KUKA KRL program: MyProgram_323().src

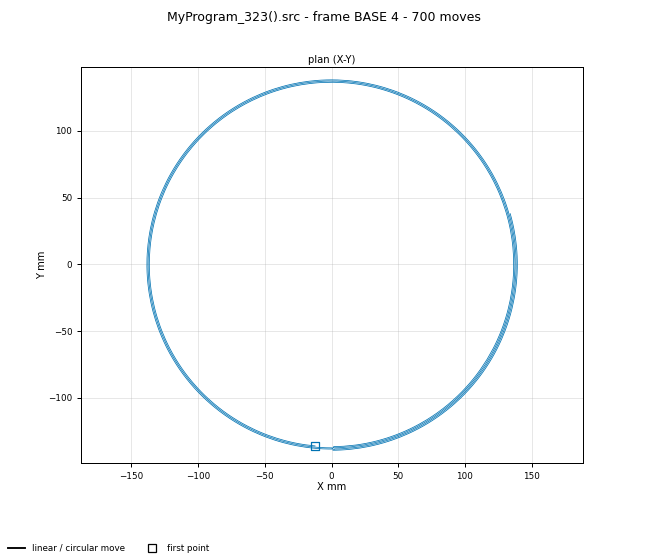
[picture p0: tool path of MyProgram_323().src in frame BASE 4, 700 of 700 moves have a stored position in this frame; points joined in program order, loops and branches not executed]
&ACCESS RVP
&REL 1
&PARAM TEMPLATE = C:\KRC\Roboter\Template\vorgabe
&PARAM EDITMASK = *
DEF MyProgram_323()
; ---- Setting reference (Base) ----
$BASE = BASE_DATA[4]

; --------------------------
; ---- Setting tool (TCP) ----
$TOOL = TOOL_DATA[3]
; --------------------------

$VEL.CP = VEL_APROX_PRINT
Startdeposition()
$VEL.CP = VEL_PRINT
LIN {X -12.3111,Y -135.9679,Z 186,A -89.4743,B 2.9889,C 0.3145,E1 2.9942,E2 182.4213} C_DIS
LIN {X -19.238,Y -135.1598,Z 186,A -92.5323,B 2.9889,C 0.3149,E1 2.9856,E2 185.4978} C_DIS
LIN {X -23.7694,Y -134.4372,Z 186,A -94.3944,B 2.9889,C 0.3139,E1 2.9805,E2 187.3522} C_DIS
LIN {X -27.1514,Y -133.7948,Z 186,A -95.8563,B 2.9889,C 0.3134,E1 2.9765,E2 188.8169} C_DIS
LIN {X -30.8353,Y -132.9948,Z 186,A -97.5736,B 2.9889,C 0.3136,E1 2.9718,E2 190.5525} C_DIS
LIN {X -35.0308,Y -131.9511,Z 186,A -99.2612,B 2.9891,C 0.3118,E1 2.9672,E2 192.2239} C_DIS
LIN {X -38.3777,Y -131.0167,Z 186,A -100.6732,B 2.9893,C 0.3107,E1 2.9634,E2 193.6301} C_DIS
LIN {X -41.0826,Y -130.1947,Z 186,A -101.9812,B 2.9893,C 0.3107,E1 2.9599,E2 194.9545} C_DIS
LIN {X -44.5379,Y -129.0528,Z 186,A -103.3999,B 2.9895,C 0.3088,E1 2.9562,E2 196.3593} C_DIS
LIN {X -47.6308,Y -127.9436,Z 186,A -104.8022,B 2.9895,C 0.3079,E1 2.9525,E2 197.7649} C_DIS
LIN {X -50.8322,Y -126.7057,Z 186,A -106.3845,B 2.9895,C 0.3074,E1 2.9483,E2 199.3662} C_DIS
LIN {X -54.0849,Y -125.3516,Z 186,A -107.898,B 2.9897,C 0.3062,E1 2.9444,E2 200.8845} C_DIS
LIN {X -57.3156,Y -123.9076,Z 186,A -109.3363,B 2.9899,C 0.3045,E1 2.9408,E2 202.3169} C_DIS
LIN {X -60.3748,Y -122.4461,Z 186,A -110.745,B 2.9901,C 0.3028,E1 2.9372,E2 203.724} C_DIS
LIN {X -63.188,Y -121.0188,Z 186,A -112.1763,B 2.9901,C 0.3019,E1 2.9336,E2 205.1695} C_DIS
LIN {X -67.1147,Y -118.8882,Z 186,A -113.9223,B 2.9905,C 0.2989,E1 2.9294,E2 206.8989} C_DIS
LIN {X -70.3666,Y -116.993,Z 186,A -115.791,B 2.9905,C 0.2985,E1 2.9248,E2 208.8057} C_DIS
LIN {X -74.0884,Y -114.6722,Z 186,A -117.6408,B 2.9908,C 0.296,E1 2.9204,E2 210.6567} C_DIS
LIN {X -77.5445,Y -112.3641,Z 186,A -119.4603,B 2.991,C 0.2938,E1 2.9162,E2 212.4861} C_DIS
LIN {X -81.1661,Y -109.7768,Z 186,A -121.4187,B 2.9912,C 0.2914,E1 2.9117,E2 214.4563} C_DIS
LIN {X -84.7687,Y -107.0191,Z 186,A -123.3765,B 2.9915,C 0.2886,E1 2.9074,E2 216.421} C_DIS
LIN {X -88.3206,Y -104.1067,Z 186,A -125.3337,B 2.9918,C 0.2855,E1 2.9032,E2 218.382} C_DIS
LIN {X -91.8517,Y -101.005,Z 186,A -127.3307,B 2.9921,C 0.2821,E1 2.899,E2 220.382} C_DIS
LIN {X -95.064,Y -97.9876,Z 186,A -129.1105,B 2.9924,C 0.2784,E1 2.8955,E2 222.1525} C_DIS
LIN {X -97.6899,Y -95.3703,Z 186,A -130.752,B 2.9927,C 0.2758,E1 2.8922,E2 223.8048} C_DIS
LIN {X -100.5401,Y -92.3602,Z 186,A -132.7985,B 2.9929,C 0.2738,E1 2.8882,E2 225.8909} C_DIS
LIN {X -103.9141,Y -88.5472,Z 186,A -134.8828,B 2.9933,C 0.2692,E1 2.8844,E2 227.9679} C_DIS
LIN {X -106.7399,Y -85.1195,Z 186,A -136.8215,B 2.9936,C 0.2656,E1 2.881,E2 229.9159} C_DIS
LIN {X -109.4795,Y -81.5656,Z 186,A -138.7616,B 2.9939,C 0.2618,E1 2.8777,E2 231.8628} C_DIS
LIN {X -112.1537,Y -77.8479,Z 186,A -140.7582,B 2.9943,C 0.2578,E1 2.8745,E2 233.8686} C_DIS
LIN {X -114.7019,Y -74.0428,Z 186,A -142.7414,B 2.9946,C 0.2537,E1 2.8714,E2 235.8592} C_DIS
LIN {X -117.0022,Y -70.3515,Z 186,A -144.5127,B 2.995,C 0.2492,E1 2.8688,E2 237.623} C_DIS
LIN {X -119.2801,Y -66.4159,Z 186,A -146.6652,B 2.9953,C 0.2456,E1 2.8658,E2 239.8061} C_DIS
LIN {X -121.5017,Y -62.2546,Z 186,A -148.7079,B 2.9957,C 0.241,E1 2.8631,E2 241.8562} C_DIS
LIN {X -123.127,Y -58.9739,Z 186,A -150.2353,B 2.996,C 0.2371,E1 2.8613,E2 243.3817} C_DIS
LIN {X -124.5737,Y -55.8532,Z 186,A -151.7312,B 2.9963,C 0.2337,E1 2.8595,E2 244.8838} C_DIS
LIN {X -125.921,Y -52.7458,Z 186,A -153.201,B 2.9965,C 0.2303,E1 2.8579,E2 246.3591} C_DIS
LIN {X -127.1093,Y -49.8151,Z 186,A -154.433,B 2.9968,C 0.2265,E1 2.8566,E2 247.5785} C_DIS
LIN {X -128.3866,Y -46.423,Z 186,A -156.1533,B 2.9971,C 0.2233,E1 2.8549,E2 249.3235} C_DIS
LIN {X -130.7067,Y -39.4242,Z 186,A -159.5632,B 2.9976,C 0.2162,E1 2.852,E2 252.7722} C_DIS
LIN {X -131.5486,Y -36.5137,Z 186,A -160.8706,B 2.9978,C 0.2129,E1 2.851,E2 254.0835} C_DIS
LIN {X -132.6266,Y -32.3816,Z 186,A -162.7159,B 2.9981,C 0.2082,E1 2.8497,E2 255.9346} C_DIS
LIN {X -133.4322,Y -28.8806,Z 186,A -164.1633,B 2.9984,C 0.2039,E1 2.8488,E2 257.3735} C_DIS
LIN {X -134.0497,Y -25.8648,Z 186,A -165.6158,B 2.9986,C 0.2009,E1 2.848,E2 258.8457} C_DIS
LIN {X -134.6734,Y -22.3906,Z 186,A -167.1966,B 2.9989,C 0.1972,E1 2.8473,E2 260.4382} C_DIS
LIN {X -135.3221,Y -18.0645,Z 186,A -169.1058,B 2.9992,C 0.1923,E1 2.8465,E2 262.3556} C_DIS
LIN {X -135.7244,Y -14.737,Z 186,A -170.6184,B 2.9994,C 0.1888,E1 2.846,E2 263.8807} C_DIS
LIN {X -136.1225,Y -10.4513,Z 186,A -172.5183,B 2.9997,C 0.184,E1 2.8456,E2 265.7912} C_DIS
LIN {X -136.3524,Y -6.8079,Z 186,A -174.1089,B 3,C 0.1799,E1 2.8453,E2 267.3882} C_DIS
LIN {X -136.4965,Y -2.6863,Z 186,A -175.9244,B 3.0002,C 0.1754,E1 2.8452,E2 269.2133} C_DIS
LIN {X -136.5203,Y 0.8769,Z 186,A -177.5554,B 3.0005,C 0.1716,E1 2.8452,E2 270.8603} C_DIS
LIN {X -136.4303,Y 5.0183,Z 186,A -179.3071,B 3.0007,C 0.1668,E1 2.8453,E2 272.6124} C_DIS
LIN {X -136.2757,Y 8.2022,Z 186,A 179.3242,B 3.0009,C 0.1631,E1 2.8455,E2 273.9841} C_DIS
LIN {X -136.0283,Y 11.6019,Z 186,A 177.7468,B 3.0011,C 0.1596,E1 2.8459,E2 275.5788} C_DIS
LIN {X -135.6057,Y 15.7966,Z 186,A 175.8905,B 3.0014,C 0.1549,E1 2.8464,E2 277.4448} C_DIS
LIN {X -135.1037,Y 19.6307,Z 186,A 174.1589,B 3.0016,C 0.1508,E1 2.8471,E2 279.1888} C_DIS
LIN {X -134.4438,Y 23.7324,Z 186,A 172.4562,B 3.0018,C 0.1458,E1 2.8479,E2 280.8851} C_DIS
LIN {X -133.8588,Y 26.8368,Z 186,A 170.5174,B 3.0018,C 0.1442,E1 2.849,E2 282.8987} C_DIS
LIN {X -132.936,Y 31.0929,Z 186,A 168.9702,B 3.0022,C 0.1382,E1 2.8499,E2 284.4101} C_DIS
LIN {X -131.9802,Y 34.9217,Z 186,A 167.2952,B 3.0024,C 0.1338,E1 2.8511,E2 286.0861} C_DIS
LIN {X -131.1717,Y 37.8484,Z 186,A 165.5608,B 3.0024,C 0.1319,E1 2.8525,E2 287.8762} C_DIS
LIN {X -129.9932,Y 41.7134,Z 186,A 164.2257,B 3.0027,C 0.1261,E1 2.8536,E2 289.1657} C_DIS
LIN {X -129.1127,Y 44.3649,Z 186,A 162.8354,B 3.0028,C 0.1238,E1 2.8548,E2 290.5819} C_DIS
LIN {X -127.3868,Y 49.1014,Z 186,A 160.7805,B 3.003,C 0.118,E1 2.8568,E2 292.6278} C_DIS
LIN {X -124.8679,Y 55.1955,Z 186,A 157.597,B 3.0033,C 0.1124,E1 2.8604,E2 295.8601} C_DIS
LIN {X -123.4731,Y 58.2496,Z 186,A 156.3105,B 3.0033,C 0.1083,E1 2.8619,E2 297.1306} C_DIS
LIN {X -121.8264,Y 61.6167,Z 186,A 154.8044,B 3.0035,C 0.1042,E1 2.8637,E2 298.6272} C_DIS
LIN {X -120.0726,Y 64.9727,Z 186,A 153.0054,B 3.0037,C 0.101,E1 2.8661,E2 300.4508} C_DIS
LIN {X -117.8522,Y 68.9177,Z 186,A 151.0476,B 3.0037,C 0.0966,E1 2.8689,E2 302.4141} C_DIS
LIN {X -115.5398,Y 72.7277,Z 186,A 149.3838,B 3.004,C 0.0914,E1 2.8713,E2 304.0513} C_DIS
LIN {X -112.8554,Y 76.8272,Z 186,A 146.5212,B 3.004,C 0.0898,E1 2.8759,E2 307.0099} C_DIS
LIN {X -110.2473,Y 80.5257,Z 186,A 144.9632,B 3.0042,C 0.0842,E1 2.8783,E2 308.5255} C_DIS
LIN {X -108.0587,Y 83.4392,Z 186,A 142.6585,B 3.0042,C 0.0839,E1 2.8825,E2 310.9221} C_DIS
LIN {X -104.259,Y 88.1412,Z 186,A 140.5187,B 3.0044,C 0.0769,E1 2.8862,E2 313.0125} C_DIS
LIN {X -101.9478,Y 90.8048,Z 186,A 139.2264,B 3.0044,C 0.0731,E1 2.8885,E2 314.2811} C_DIS
LIN {X -98.977,Y 94.0341,Z 186,A 137.3781,B 3.0045,C 0.0695,E1 2.8921,E2 316.1288} C_DIS
LIN {X -95.5224,Y 97.5407,Z 186,A 135.1953,B 3.0046,C 0.066,E1 2.8964,E2 318.3242} C_DIS
LIN {X -92.1681,Y 100.7167,Z 186,A 133.1879,B 3.0046,C 0.0627,E1 2.9005,E2 320.3384} C_DIS
LIN {X -88.7865,Y 103.7103,Z 186,A 131.2058,B 3.0048,C 0.0597,E1 2.9047,E2 322.3296} C_DIS
LIN {X -86.4597,Y 105.6572,Z 186,A 129.1909,B 3.0048,C 0.0608,E1 2.9093,E2 324.4318} C_DIS
LIN {X -81.7175,Y 109.3665,Z 186,A 127.307,B 3.0048,C 0.0538,E1 2.9133,E2 326.2376} C_DIS
LIN {X -78.0842,Y 111.9893,Z 186,A 125.4022,B 3.0049,C 0.051,E1 2.9176,E2 328.1439} C_DIS
LIN {X -74.4651,Y 114.4277,Z 186,A 123.4234,B 3.0049,C 0.049,E1 2.9223,E2 330.139} C_DIS
LIN {X -69.1963,Y 117.6886,Z 186,A 120.8537,B 3.005,C 0.0453,E1 2.9284,E2 332.7033} C_DIS
LIN {X -64.6844,Y 120.2276,Z 186,A 117.9757,B 3.005,C 0.046,E1 2.9357,E2 335.6634} C_DIS
LIN {X -59.6478,Y 122.8047,Z 186,A 116.2676,B 3.005,C 0.04,E1 2.9398,E2 337.2911} C_DIS
LIN {X -56.2549,Y 124.394,Z 186,A 114.6333,B 3.0051,C 0.0386,E1 2.9439,E2 338.9317} C_DIS
LIN {X -53.3798,Y 125.6562,Z 186,A 112.5963,B 3.0051,C 0.041,E1 2.9494,E2 341.0531} C_DIS
LIN {X -48.161,Y 127.745,Z 186,A 110.9689,B 3.0051,C 0.035,E1 2.9534,E2 342.5924} C_DIS
LIN {X -44.7133,Y 128.9919,Z 186,A 109.423,B 3.0051,C 0.0338,E1 2.9575,E2 344.1382} C_DIS
LIN {X -41.5386,Y 130.0491,Z 186,A 108.0354,B 3.0051,C 0.0326,E1 2.9612,E2 345.523} C_DIS
LIN {X -37.3561,Y 131.313,Z 186,A 105.9999,B 3.0051,C 0.0325,E1 2.9667,E2 347.5815} C_DIS
LIN {X -33.3708,Y 132.3808,Z 186,A 104.3549,B 3.0051,C 0.031,E1 2.9711,E2 349.2152} C_DIS
LIN {X -29.3101,Y 133.3395,Z 186,A 102.5381,B 3.0051,C 0.0305,E1 2.9761,E2 351.0389} C_DIS
LIN {X -25.8157,Y 134.0591,Z 186,A 101.1794,B 3.0052,C 0.029,E1 2.9798,E2 352.3802} C_DIS
LIN {X -22.6569,Y 134.629,Z 186,A 99.7557,B 3.0052,C 0.029,E1 2.9837,E2 353.8124} C_DIS
LIN {X -19.1156,Y 135.1773,Z 186,A 98.1668,B 3.0052,C 0.029,E1 2.9881,E2 355.4106} C_DIS
LIN {X -15.9064,Y 135.5925,Z 186,A 96.2554,B 3.0052,C 0.0321,E1 2.9936,E2 357.3868} C_DIS
LIN {X -10.8726,Y 136.0899,Z 186,A 94.9122,B 3.0052,C 0.0271,E1 2.9971,E2 358.6368} C_DIS
LIN {X -6.7864,Y 136.3535,Z 186,A 92.9753,B 3.0052,C 0.0284,E1 3.0026,E2 360.5989} C_DIS
LIN {X 1.2265,Y 136.5176,Z 186,A 89.7328,B 3.0052,C 0.0279,E1 3.0116,E2 363.8257} C_DIS
LIN {X 7.1604,Y 136.3347,Z 186,A 87.0766,B 3.0052,C 0.0296,E1 3.0191,E2 366.5005} C_DIS
LIN {X 12.8357,Y 135.9176,Z 186,A 84.5619,B 3.0052,C 0.0312,E1 3.0261,E2 369.0293} C_DIS
LIN {X 18.3432,Y 135.2855,Z 186,A 82.3763,B 3.0052,C 0.0314,E1 3.0321,E2 371.1974} C_DIS
LIN {X 22.0077,Y 134.7373,Z 186,A 80.9108,B 3.0052,C 0.0316,E1 3.0361,E2 372.6518} C_DIS
LIN {X 25.5439,Y 134.111,Z 186,A 79.4605,B 3.0052,C 0.0322,E1 3.0401,E2 374.0947} C_DIS
LIN {X 29.2124,Y 133.3606,Z 186,A 77.8146,B 3.0052,C 0.0338,E1 3.0446,E2 375.749} C_DIS
LIN {X 33.2752,Y 132.405,Z 186,A 76.1571,B 3.0052,C 0.0345,E1 3.0491,E2 377.3949} C_DIS
LIN {X 36.6894,Y 131.4995,Z 186,A 74.7084,B 3.0052,C 0.0355,E1 3.053,E2 378.8391} C_DIS
LIN {X 40.0511,Y 130.5149,Z 186,A 73.3177,B 3.0052,C 0.0363,E1 3.0567,E2 380.22} C_DIS
LIN {X 43.289,Y 129.477,Z 186,A 71.8669,B 3.0052,C 0.0379,E1 3.0606,E2 381.6734} C_DIS
LIN {X 46.795,Y 128.2525,Z 186,A 70.2657,B 3.0051,C 0.0399,E1 3.0648,E2 383.2794} C_DIS
LIN {X 50.596,Y 126.8009,Z 186,A 68.7271,B 3.0051,C 0.0405,E1 3.0687,E2 384.7975} C_DIS
LIN {X 53.9337,Y 125.4169,Z 186,A 67.2445,B 3.0051,C 0.0421,E1 3.0726,E2 386.2757} C_DIS
LIN {X 57.0285,Y 124.0404,Z 186,A 65.7416,B 3.0051,C 0.0445,E1 3.0764,E2 387.7883} C_DIS
LIN {X 60.1298,Y 122.5669,Z 186,A 64.3487,B 3.005,C 0.046,E1 3.0799,E2 389.1752} C_DIS
LIN {X 63.3023,Y 120.9587,Z 186,A 62.9182,B 3.005,C 0.0476,E1 3.0834,E2 390.5981} C_DIS
LIN {X 67.5166,Y 118.6603,Z 186,A 60.8638,B 3.005,C 0.0509,E1 3.0885,E2 392.6573} C_DIS
LIN {X 71.4257,Y 116.349,Z 186,A 59.0755,B 3.0049,C 0.0529,E1 3.0927,E2 394.4313} C_DIS
LIN {X 74.975,Y 114.0942,Z 186,A 57.2858,B 3.0049,C 0.0559,E1 3.0969,E2 396.224} C_DIS
LIN {X 78.8427,Y 111.4566,Z 186,A 55.4054,B 3.0048,C 0.0585,E1 3.1012,E2 398.0942} C_DIS
LIN {X 82.5066,Y 108.7726,Z 186,A 53.5229,B 3.0048,C 0.0617,E1 3.1054,E2 399.9739} C_DIS
LIN {X 86.0456,Y 105.9956,Z 186,A 51.6692,B 3.0047,C 0.0649,E1 3.1095,E2 401.8236} C_DIS
LIN {X 89.4469,Y 103.1414,Z 186,A 49.8729,B 3.0046,C 0.0678,E1 3.1133,E2 403.6119} C_DIS
LIN {X 95.1093,Y 97.9437,Z 186,A 46.7896,B 3.0045,C 0.073,E1 3.1196,E2 406.6783} C_DIS
LIN {X 97.8786,Y 95.1766,Z 186,A 44.8441,B 3.0043,C 0.079,E1 3.1234,E2 408.6608} C_DIS
LIN {X 100.6933,Y 92.1935,Z 186,A 43.5559,B 3.0043,C 0.0789,E1 3.1258,E2 409.8967} C_DIS
LIN {X 103.6368,Y 88.8719,Z 186,A 41.7233,B 3.0043,C 0.0827,E1 3.1291,E2 411.7259} C_DIS
LIN {X 106.4156,Y 85.5248,Z 186,A 39.9701,B 3.0041,C 0.0861,E1 3.1322,E2 413.4707} C_DIS
LIN {X 109.1359,Y 82.0252,Z 186,A 38.179,B 3.0041,C 0.0897,E1 3.1352,E2 415.2538} C_DIS
LIN {X 111.7542,Y 78.4208,Z 186,A 36.3595,B 3.0039,C 0.0936,E1 3.1382,E2 417.0677} C_DIS
LIN {X 113.7016,Y 75.5694,Z 186,A 34.9815,B 3.0039,C 0.0964,E1 3.1403,E2 418.4373} C_DIS
LIN {X 116.1565,Y 71.7395,Z 186,A 32.9663,B 3.0036,C 0.102,E1 3.1433,E2 420.4662} C_DIS
LIN {X 119.222,Y 66.5209,Z 186,A 30.6725,B 3.0035,C 0.106,E1 3.1465,E2 422.7306} C_DIS
LIN {X 121.467,Y 62.3227,Z 186,A 28.9267,B 3.0034,C 0.1087,E1 3.1487,E2 424.4458} C_DIS
LIN {X 123.0445,Y 59.1467,Z 186,A 27.6386,B 3.0034,C 0.1106,E1 3.1503,E2 425.7097} C_DIS
LIN {X 124.2101,Y 56.6613,Z 186,A 26.2314,B 3.0031,C 0.116,E1 3.152,E2 427.1491} C_DIS
LIN {X 125.8549,Y 52.904,Z 186,A 24.7918,B 3.0031,C 0.1178,E1 3.1535,E2 428.5544} C_DIS
LIN {X 128.2307,Y 46.8553,Z 186,A 22.0445,B 3.0027,C 0.1252,E1 3.1563,E2 431.3054} C_DIS
LIN {X 129.4084,Y 43.4949,Z 186,A 20.6357,B 3.0027,C 0.1284,E1 3.1575,E2 432.7043} C_DIS
LIN {X 130.4095,Y 40.3955,Z 186,A 19.2687,B 3.0024,C 0.1321,E1 3.1587,E2 434.0719} C_DIS
LIN {X 131.4793,Y 36.7617,Z 186,A 17.7861,B 3.0024,C 0.1354,E1 3.1598,E2 435.542} C_DIS
LIN {X 132.5414,Y 32.7352,Z 186,A 16.0718,B 3.0021,C 0.1398,E1 3.161,E2 437.2531} C_DIS
LIN {X 133.3882,Y 29.0848,Z 186,A 14.6294,B 3.002,C 0.1429,E1 3.1619,E2 438.68} C_DIS
LIN {X 134.1341,Y 25.4233,Z 186,A 13.1458,B 3.0018,C 0.1464,E1 3.1627,E2 440.1538} C_DIS
LIN {X 134.8123,Y 21.5488,Z 186,A 11.5791,B 3.0016,C 0.1502,E1 3.1634,E2 441.7109} C_DIS
LIN {X 135.2752,Y 18.422,Z 186,A 9.6378,B 3.0011,C 0.1599,E1 3.1642,E2 443.7298} C_DIS
LIN {X 135.9042,Y 12.9748,Z 186,A 8.4515,B 3.0013,C 0.1555,E1 3.1645,E2 444.7776} C_DIS
LIN {X 136.407,Y 5.6162,Z 186,A 5.3662,B 3.0009,C 0.1642,E1 3.1651,E2 447.8638} C_DIS
LIN {X 136.5062,Y -2.0993,Z 186,A 1.3136,B 2.9999,C 0.1812,E1 3.1651,E2 452.0211} C_DIS
LIN {X 136.2808,Y -8.1196,Z 186,A -0.3193,B 2.9999,C 0.1796,E1 3.1648,E2 453.5429} C_DIS
LIN {X 135.9648,Y -12.3354,Z 186,A -2.5049,B 2.9994,C 0.1886,E1 3.1643,E2 455.7818} C_DIS
LIN {X 135.4992,Y -16.6892,Z 186,A -3.8904,B 2.9994,C 0.1894,E1 3.1639,E2 457.1113} C_DIS
LIN {X 134.9309,Y -20.7833,Z 186,A -5.4477,B 2.9992,C 0.1925,E1 3.1632,E2 458.6473} C_DIS
LIN {X 134.3821,Y -24.0773,Z 186,A -6.7467,B 2.999,C 0.1954,E1 3.1626,E2 459.9342} C_DIS
LIN {X 133.7801,Y -27.2236,Z 186,A -7.9962,B 2.9988,C 0.1982,E1 3.162,E2 461.1726} C_DIS
LIN {X 133.149,Y -30.1605,Z 186,A -9.288,B 2.9986,C 0.202,E1 3.1612,E2 462.4692} C_DIS
LIN {X 132.4036,Y -33.2808,Z 186,A -10.5452,B 2.9984,C 0.2048,E1 3.1604,E2 463.716} C_DIS
LIN {X 131.556,Y -36.4873,Z 186,A -11.9479,B 2.9981,C 0.2087,E1 3.1593,E2 465.1211} C_DIS
LIN {X 130.4126,Y -40.3853,Z 186,A -13.5042,B 2.9979,C 0.2119,E1 3.1581,E2 466.6597} C_DIS
LIN {X 128.6481,Y -45.6978,Z 186,A -15.827,B 2.9974,C 0.218,E1 3.156,E2 468.981} C_DIS
LIN {X 127.2845,Y -49.3646,Z 186,A -17.2732,B 2.9973,C 0.2204,E1 3.1546,E2 470.4032} C_DIS
LIN {X 125.978,Y -52.6091,Z 186,A -18.8924,B 2.9969,C 0.2258,E1 3.1529,E2 472.043} C_DIS
LIN {X 124.0407,Y -57.0278,Z 186,A -20.7104,B 2.9966,C 0.229,E1 3.1508,E2 473.8359} C_DIS
LIN {X 122.5799,Y -60.1036,Z 186,A -22.0566,B 2.9964,C 0.2319,E1 3.1492,E2 475.1725} C_DIS
LIN {X 120.9462,Y -63.3261,Z 186,A -23.2628,B 2.9964,C 0.2328,E1 3.1477,E2 476.3398} C_DIS
LIN {X 116.5433,Y -71.109,Z 186,A -27.0396,B 2.9956,C 0.2424,E1 3.1425,E2 480.123} C_DIS
LIN {X 111.4881,Y -78.7982,Z 186,A -30.8987,B 2.9948,C 0.2517,E1 3.1365,E2 483.985} C_DIS
LIN {X 108.7858,Y -82.4892,Z 186,A -32.7657,B 2.9945,C 0.2556,E1 3.1334,E2 485.8467} C_DIS
LIN {X 106.2159,Y -85.7725,Z 186,A -34.4538,B 2.9942,C 0.259,E1 3.1305,E2 487.5282} C_DIS
LIN {X 103.4473,Y -89.0919,Z 186,A -36.1448,B 2.9939,C 0.2619,E1 3.1274,E2 489.2046} C_DIS
LIN {X 100.2325,Y -92.6949,Z 186,A -38.1537,B 2.9936,C 0.2662,E1 3.1237,E2 491.2128} C_DIS
LIN {X 97.6082,Y -95.4536,Z 186,A -40.0748,B 2.993,C 0.2725,E1 3.1199,E2 493.1773} C_DIS
LIN {X 94.4964,Y -98.5353,Z 186,A -41.3875,B 2.993,C 0.2715,E1 3.1174,E2 494.423} C_DIS
LIN {X 90.4497,Y -102.2623,Z 186,A -43.6905,B 2.9927,C 0.276,E1 3.1126,E2 496.7271} C_DIS
LIN {X 87.1048,Y -105.126,Z 186,A -45.9044,B 2.992,C 0.2828,E1 3.1077,E2 498.9902} C_DIS
LIN {X 83.5684,Y -107.9586,Z 186,A -46.982,B 2.9924,C 0.279,E1 3.1056,E2 499.9614} C_DIS
LIN {X 79.133,Y -111.2511,Z 186,A -49.5837,B 2.9918,C 0.2856,E1 3.0997,E2 502.6023} C_DIS
LIN {X 75.5393,Y -113.7217,Z 186,A -51.357,B 2.9915,C 0.2882,E1 3.0956,E2 504.3694} C_DIS
LIN {X 71.532,Y -116.2838,Z 186,A -53.3903,B 2.9912,C 0.2918,E1 3.0907,E2 506.4091} C_DIS
LIN {X 65.5581,Y -119.7535,Z 186,A -56.1325,B 2.9909,C 0.2949,E1 3.0841,E2 509.1329} C_DIS
LIN {X 62.147,Y -121.5565,Z 186,A -57.6033,B 2.9908,C 0.2959,E1 3.0805,E2 510.5852} C_DIS
LIN {X 59.1591,Y -123.0385,Z 186,A -59.0602,B 2.9905,C 0.2983,E1 3.0768,E2 512.0506} C_DIS
LIN {X 55.5909,Y -124.6911,Z 186,A -60.5881,B 2.9905,C 0.2995,E1 3.073,E2 513.5636} C_DIS
LIN {X 52.4141,Y -126.0595,Z 186,A -62.034,B 2.9902,C 0.3012,E1 3.0693,E2 515.0097} C_DIS
LIN {X 48.6609,Y -127.5578,Z 186,A -63.681,B 2.9901,C 0.3028,E1 3.065,E2 516.6515} C_DIS
LIN {X 44.8703,Y -128.9375,Z 186,A -65.3992,B 2.9899,C 0.3049,E1 3.0605,E2 518.374} C_DIS
LIN {X 41.2755,Y -130.1331,Z 186,A -66.9553,B 2.9897,C 0.3062,E1 3.0563,E2 519.9268} C_DIS
LIN {X 37.195,Y -131.3581,Z 186,A -68.7222,B 2.9896,C 0.3077,E1 3.0516,E2 521.6921} C_DIS
LIN {X 33.8183,Y -132.2672,Z 186,A -70.1741,B 2.9894,C 0.3089,E1 3.0477,E2 523.1427} C_DIS
LIN {X 30.2259,Y -133.134,Z 186,A -71.6818,B 2.9894,C 0.3098,E1 3.0436,E2 524.6457} C_DIS
LIN {X 25.9781,Y -134.028,Z 186,A -73.3502,B 2.9894,C 0.31,E1 3.0391,E2 526.2949} C_DIS
LIN {X 21.4124,Y -134.8332,Z 186,A -75.69,B 2.9889,C 0.3142,E1 3.0325,E2 528.6879} C_DIS
LIN {X 18.0587,Y -135.3228,Z 186,A -76.8354,B 2.989,C 0.3129,E1 3.0294,E2 529.7976} C_DIS
LIN {X 9.0374,Y -136.2243,Z 186,A -80.7077,B 2.9888,C 0.315,E1 3.0186,E2 533.6809} C_DIS
LIN {X 1.6488,Y -136.5137,Z 186,A -83.7384,B 2.9888,C 0.3153,E1 3.0101,E2 536.7035} C_DIS
LIN {X 1.6488,Y -136.5137,Z 186,A -83.7384,B 2.9888,C 0.3153,E1 3.0101,E2 536.7035} C_DIS
Enddeposition()
LIN {X 0.9838,Y -137.4158,Z 186,A -83.4566,B 2.9647,C 0.3121,E1 2.9867,E2 536.3846} C_DIS
Startdeposition()
$VEL.CP = VEL_PRINT
LIN {X 6.0843,Y -137.2888,Z 186,A -80.8856,B 2.9651,C 0.3083,E1 2.9941,E2 533.7529} C_DIS
LIN {X 15.2711,Y -136.572,Z 186,A -77.5006,B 2.9649,C 0.3101,E1 3.0034,E2 530.4276} C_DIS
LIN {X 23.8245,Y -135.3415,Z 186,A -73.9161,B 2.9651,C 0.3082,E1 3.0133,E2 526.844} C_DIS
LIN {X 27.9411,Y -134.5524,Z 186,A -72.0646,B 2.9654,C 0.3062,E1 3.0184,E2 524.9774} C_DIS
LIN {X 30.6359,Y -133.9634,Z 186,A -70.8892,B 2.9654,C 0.3051,E1 3.0216,E2 523.7979} C_DIS
LIN {X 33.9603,Y -133.1595,Z 186,A -69.4585,B 2.9656,C 0.3038,E1 3.0255,E2 522.3656} C_DIS
LIN {X 37.3207,Y -132.2573,Z 186,A -68.0274,B 2.9657,C 0.3027,E1 3.0293,E2 520.9363} C_DIS
LIN {X 41.0982,Y -131.1344,Z 186,A -66.3318,B 2.9659,C 0.3006,E1 3.0339,E2 519.2326} C_DIS
LIN {X 45.8226,Y -129.559,Z 186,A -64.2508,B 2.9661,C 0.2984,E1 3.0394,E2 517.1496} C_DIS
LIN {X 49.2855,Y -128.2807,Z 186,A -62.9983,B 2.9661,C 0.299,E1 3.0426,E2 515.9346} C_DIS
LIN {X 51.8725,Y -127.2565,Z 186,A -61.7597,B 2.9663,C 0.2969,E1 3.0458,E2 514.6847} C_DIS
LIN {X 54.8322,Y -126.0088,Z 186,A -60.3926,B 2.9665,C 0.295,E1 3.0494,E2 513.3128} C_DIS
LIN {X 58.2534,Y -124.4653,Z 186,A -58.9074,B 2.9666,C 0.2936,E1 3.0531,E2 511.8373} C_DIS
LIN {X 60.9886,Y -123.1467,Z 186,A -57.6529,B 2.9668,C 0.292,E1 3.0562,E2 510.5833} C_DIS
LIN {X 64.5773,Y -121.3054,Z 186,A -56.0289,B 2.967,C 0.2901,E1 3.0603,E2 508.9659} C_DIS
LIN {X 71.2749,Y -117.4953,Z 186,A -53.0145,B 2.9673,C 0.2869,E1 3.0675,E2 505.9759} C_DIS
LIN {X 73.8968,Y -115.8643,Z 186,A -51.6077,B 2.9676,C 0.2837,E1 3.0709,E2 504.5521} C_DIS
LIN {X 77.4136,Y -113.5454,Z 186,A -49.8532,B 2.9679,C 0.2808,E1 3.0749,E2 502.7966} C_DIS
LIN {X 81.4654,Y -110.6736,Z 186,A -47.8505,B 2.9681,C 0.2777,E1 3.0795,E2 500.8014} C_DIS
LIN {X 85.1177,Y -107.8902,Z 186,A -45.9085,B 2.9685,C 0.274,E1 3.0838,E2 498.8543} C_DIS
LIN {X 88.7967,Y -104.883,Z 186,A -44.0465,B 2.9687,C 0.2713,E1 3.0877,E2 497.0066} C_DIS
LIN {X 92.6493,Y -101.4962,Z 186,A -41.9771,B 2.9691,C 0.2677,E1 3.092,E2 494.9448} C_DIS
LIN {X 95.8665,Y -98.4631,Z 186,A -40.0732,B 2.9695,C 0.2634,E1 3.0959,E2 493.0313} C_DIS
LIN {X 99.4539,Y -94.8376,Z 186,A -38.1905,B 2.9696,C 0.2612,E1 3.0995,E2 491.1796} C_DIS
LIN {X 103.7571,Y -90.1099,Z 186,A -35.8146,B 2.9699,C 0.2581,E1 3.1039,E2 488.84} C_DIS
LIN {X 106.2348,Y -87.175,Z 186,A -34.2526,B 2.9702,C 0.2549,E1 3.1067,E2 487.282} C_DIS
LIN {X 108.3221,Y -84.5678,Z 186,A -32.6836,B 2.9706,C 0.25,E1 3.1094,E2 485.6885} C_DIS
LIN {X 111.0315,Y -80.9778,Z 186,A -30.8633,B 2.9709,C 0.2462,E1 3.1124,E2 483.874} C_DIS
LIN {X 114.6998,Y -75.6916,Z 186,A -28.4907,B 2.9712,C 0.2427,E1 3.1161,E2 481.5404} C_DIS
LIN {X 116.4675,Y -72.9433,Z 186,A -27.0097,B 2.9716,C 0.2383,E1 3.1183,E2 480.0426} C_DIS
LIN {X 118.7531,Y -69.1597,Z 186,A -24.905,B 2.9721,C 0.2312,E1 3.1214,E2 477.9017} C_DIS
LIN {X 120.7699,Y -65.5739,Z 186,A -23.8905,B 2.9719,C 0.2337,E1 3.1226,E2 476.9785} C_DIS
LIN {X 122.7353,Y -61.8148,Z 186,A -22.0061,B 2.9724,C 0.2281,E1 3.1251,E2 475.0774} C_DIS
LIN {X 124.2064,Y -58.8022,Z 186,A -20.6294,B 2.9726,C 0.2247,E1 3.1267,E2 473.7024} C_DIS
LIN {X 126.0715,Y -54.6872,Z 186,A -18.8431,B 2.9729,C 0.2207,E1 3.1287,E2 471.9275} C_DIS
LIN {X 127.5288,Y -51.197,Z 186,A -17.3304,B 2.9732,C 0.2172,E1 3.1303,E2 470.422} C_DIS
LIN {X 128.6557,Y -48.2952,Z 186,A -16.0219,B 2.9734,C 0.2136,E1 3.1316,E2 469.111} C_DIS
LIN {X 130.0508,Y -44.4062,Z 186,A -14.3731,B 2.9737,C 0.2097,E1 3.1331,E2 467.4707} C_DIS
LIN {X 131.4625,Y -40.0296,Z 186,A -12.6229,B 2.974,C 0.2062,E1 3.1346,E2 465.7409} C_DIS
LIN {X 132.399,Y -36.814,Z 186,A -11.256,B 2.9742,C 0.2026,E1 3.1356,E2 464.3768} C_DIS
LIN {X 133.3831,Y -33.0796,Z 186,A -9.6115,B 2.9745,C 0.1979,E1 3.1368,E2 462.7267} C_DIS
LIN {X 134.3729,Y -28.7877,Z 186,A -7.9633,B 2.9747,C 0.1947,E1 3.1378,E2 461.1016} C_DIS
LIN {X 134.9919,Y -25.7283,Z 186,A -6.7307,B 2.9749,C 0.1917,E1 3.1384,E2 459.8771} C_DIS
LIN {X 135.5919,Y -22.3538,Z 186,A -5.3512,B 2.9752,C 0.1882,E1 3.1391,E2 458.5029} C_DIS
LIN {X 136.5249,Y -15.6875,Z 186,A -2.7552,B 2.9755,C 0.1825,E1 3.14,E2 455.9325} C_DIS
LIN {X 136.7964,Y -13.0983,Z 186,A -1.6644,B 2.9757,C 0.1794,E1 3.1403,E2 454.8402} C_DIS
LIN {X 137.1107,Y -9.2737,Z 186,A 0.0096,B 2.976,C 0.1741,E1 3.1407,E2 453.1555} C_DIS
LIN {X 137.3982,Y -2.5811,Z 186,A 2.7871,B 2.9765,C 0.1664,E1 3.1409,E2 450.3782} C_DIS
LIN {X 137.4216,Y 0.6595,Z 186,A 3.8367,B 2.9765,C 0.1656,E1 3.1409,E2 449.3667} C_DIS
LIN {X 137.3626,Y 4.0518,Z 186,A 5.1748,B 2.9767,C 0.1623,E1 3.1409,E2 448.0376} C_DIS
LIN {X 136.9597,Y 11.2669,Z 186,A 7.8516,B 2.977,C 0.1572,E1 3.1404,E2 445.4023} C_DIS
LIN {X 136.6432,Y 14.6094,Z 186,A 9.9047,B 2.9775,C 0.1468,E1 3.1398,E2 443.2642} C_DIS
LIN {X 136.065,Y 19.2645,Z 186,A 11.2095,B 2.9775,C 0.1478,E1 3.1393,E2 442.0422} C_DIS
LIN {X 135.5475,Y 22.6197,Z 186,A 12.6125,B 2.9776,C 0.1439,E1 3.1387,E2 440.6399} C_DIS
LIN {X 134.9367,Y 26.0175,Z 186,A 14.0063,B 2.9778,C 0.1404,E1 3.138,E2 439.2512} C_DIS
LIN {X 134.2553,Y 29.3323,Z 186,A 15.2719,B 2.9779,C 0.1379,E1 3.1372,E2 438.0034} C_DIS
LIN {X 133.6055,Y 32.1607,Z 186,A 16.4676,B 2.9781,C 0.1347,E1 3.1365,E2 436.8089} C_DIS
LIN {X 132.7591,Y 35.493,Z 186,A 17.8355,B 2.9782,C 0.1314,E1 3.1355,E2 435.4486} C_DIS
LIN {X 131.7553,Y 39.0576,Z 186,A 19.3108,B 2.9784,C 0.1279,E1 3.1344,E2 433.9813} C_DIS
LIN {X 130.7895,Y 42.1778,Z 186,A 20.6176,B 2.9784,C 0.1248,E1 3.1333,E2 432.6809} C_DIS
LIN {X 129.6667,Y 45.5141,Z 186,A 22.0449,B 2.9786,C 0.1212,E1 3.132,E2 431.258} C_DIS
LIN {X 126.5434,Y 53.5904,Z 186,A 25.9338,B 2.9791,C 0.1091,E1 3.1279,E2 427.3323} C_DIS
LIN {X 124.8673,Y 57.3841,Z 186,A 26.9568,B 2.9791,C 0.1113,E1 3.1269,E2 426.398} C_DIS
LIN {X 123.7691,Y 59.7174,Z 186,A 28.1707,B 2.9791,C 0.1072,E1 3.1254,E2 425.1663} C_DIS
LIN {X 122.2036,Y 62.8593,Z 186,A 29.6968,B 2.9793,C 0.1029,E1 3.1234,E2 423.6317} C_DIS
LIN {X 119.9741,Y 67.0193,Z 186,A 32.3442,B 2.9797,C 0.0917,E1 3.1197,E2 420.8975} C_DIS
LIN {X 116.5838,Y 72.7563,Z 186,A 33.7718,B 2.9795,C 0.0975,E1 3.1179,E2 419.6397} C_DIS
LIN {X 114.503,Y 75.9897,Z 186,A 35.7658,B 2.9797,C 0.09,E1 3.1148,E2 417.5963} C_DIS
LIN {X 112.067,Y 79.5386,Z 186,A 37.463,B 2.9798,C 0.0867,E1 3.1121,E2 415.9109} C_DIS
LIN {X 109.5431,Y 82.9795,Z 186,A 39.1912,B 2.9799,C 0.0831,E1 3.1092,E2 414.1886} C_DIS
LIN {X 106.7921,Y 86.4913,Z 186,A 40.9872,B 2.98,C 0.0795,E1 3.1061,E2 412.4002} C_DIS
LIN {X 104.1696,Y 89.6322,Z 186,A 42.6346,B 2.9801,C 0.0762,E1 3.1031,E2 410.7597} C_DIS
LIN {X 100.9305,Y 93.2651,Z 186,A 44.5232,B 2.9802,C 0.0732,E1 3.0996,E2 408.8883} C_DIS
LIN {X 98.2197,Y 96.1153,Z 186,A 46.1373,B 2.9802,C 0.07,E1 3.0965,E2 407.2772} C_DIS
LIN {X 95.1885,Y 99.1186,Z 186,A 47.8582,B 2.9804,C 0.0669,E1 3.093,E2 405.5633} C_DIS
LIN {X 91.7583,Y 102.3017,Z 186,A 49.558,B 2.9804,C 0.0652,E1 3.0896,E2 403.8944} C_DIS
LIN {X 89.3603,Y 104.4038,Z 186,A 51.1089,B 2.9804,C 0.0608,E1 3.0863,E2 402.316} C_DIS
LIN {X 85.8159,Y 107.3357,Z 186,A 52.8856,B 2.9805,C 0.0584,E1 3.0825,E2 400.5566} C_DIS
LIN {X 82.4493,Y 109.9432,Z 186,A 54.6776,B 2.9805,C 0.0551,E1 3.0785,E2 398.7625} C_DIS
LIN {X 78.8178,Y 112.5751,Z 186,A 56.5042,B 2.9806,C 0.0523,E1 3.0743,E2 396.9413} C_DIS
LIN {X 75.1176,Y 115.0769,Z 186,A 58.3031,B 2.9806,C 0.0497,E1 3.0701,E2 395.1502} C_DIS
LIN {X 71.316,Y 117.4705,Z 186,A 60.1218,B 2.9807,C 0.0472,E1 3.0658,E2 393.3383} C_DIS
LIN {X 67.4421,Y 119.7364,Z 186,A 61.9404,B 2.9807,C 0.0449,E1 3.0614,E2 391.5262} C_DIS
LIN {X 63.4637,Y 121.8903,Z 186,A 63.7342,B 2.9807,C 0.0429,E1 3.057,E2 389.7439} C_DIS
LIN {X 60.2709,Y 123.5008,Z 186,A 65.1211,B 2.9808,C 0.0417,E1 3.0536,E2 388.37} C_DIS
LIN {X 57.5507,Y 124.7903,Z 186,A 66.3847,B 2.9808,C 0.04,E1 3.0504,E2 387.1054} C_DIS
LIN {X 54.3365,Y 126.2231,Z 186,A 67.7706,B 2.9808,C 0.0389,E1 3.0469,E2 385.7297} C_DIS
LIN {X 51.1948,Y 127.5297,Z 186,A 69.1505,B 2.9808,C 0.0375,E1 3.0433,E2 384.3547} C_DIS
LIN {X 47.9965,Y 128.7676,Z 186,A 70.629,B 2.9808,C 0.0355,E1 3.0394,E2 382.8706} C_DIS
LIN {X 44.8342,Y 129.9024,Z 186,A 71.9575,B 2.9808,C 0.0346,E1 3.036,E2 381.5512} C_DIS
LIN {X 41.6668,Y 130.9528,Z 186,A 73.3603,B 2.9809,C 0.0332,E1 3.0322,E2 380.1473} C_DIS
LIN {X 38.2882,Y 131.9805,Z 186,A 74.7663,B 2.9809,C 0.0323,E1 3.0285,E2 378.7497} C_DIS
LIN {X 35.1184,Y 132.859,Z 186,A 76.1537,B 2.9809,C 0.031,E1 3.0247,E2 377.3608} C_DIS
LIN {X 31.2605,Y 133.8207,Z 186,A 77.8882,B 2.9809,C 0.0292,E1 3.02,E2 375.6174} C_DIS
LIN {X 27.3053,Y 134.6818,Z 186,A 79.4697,B 2.9809,C 0.0288,E1 3.0157,E2 374.0492} C_DIS
LIN {X 23.9294,Y 135.3227,Z 186,A 80.8742,B 2.9809,C 0.0281,E1 3.0118,E2 372.6486} C_DIS
LIN {X 19.779,Y 135.9915,Z 186,A 83.0929,B 2.981,C 0.0239,E1 3.0056,E2 370.3735} C_DIS
LIN {X 15.3734,Y 136.561,Z 186,A 84.6616,B 2.981,C 0.025,E1 3.0013,E2 368.8402} C_DIS
LIN {X 11.324,Y 136.9549,Z 186,A 86.1675,B 2.981,C 0.0256,E1 2.9972,E2 367.3581} C_DIS
LIN {X 3.7298,Y 137.3715,Z 186,A 89.307,B 2.981,C 0.025,E1 2.9884,E2 364.2238} C_DIS
LIN {X -2.396,Y 137.4013,Z 186,A 91.829,B 2.981,C 0.025,E1 2.9814,E2 361.7068} C_DIS
LIN {X -6.3791,Y 137.2749,Z 186,A 94.4143,B 2.981,C 0.019,E1 2.9739,E2 359.0091} C_DIS
LIN {X -12.9774,Y 136.808,Z 186,A 96.4416,B 2.981,C 0.0239,E1 2.9685,E2 357.0729} C_DIS
LIN {X -16.8139,Y 136.3905,Z 186,A 97.8218,B 2.981,C 0.0257,E1 2.9647,E2 355.7214} C_DIS
LIN {X -19.8051,Y 135.9878,Z 186,A 99.191,B 2.981,C 0.0253,E1 2.9609,E2 354.3394} C_DIS
LIN {X -24.0174,Y 135.3069,Z 186,A 100.9628,B 2.981,C 0.026,E1 2.956,E2 352.5693} C_DIS
LIN {X -27.6242,Y 134.6169,Z 186,A 102.5013,B 2.981,C 0.0266,E1 2.9518,E2 351.0307} C_DIS
LIN {X -30.9424,Y 133.8934,Z 186,A 103.8661,B 2.981,C 0.0276,E1 2.9481,E2 349.673} C_DIS
LIN {X -34.1956,Y 133.0998,Z 186,A 105.3671,B 2.981,C 0.0278,E1 2.944,E2 348.16} C_DIS
LIN {X -38.7038,Y 131.8588,Z 186,A 107.2718,B 2.981,C 0.0293,E1 2.9389,E2 346.2618} C_DIS
LIN {X -41.9591,Y 130.8594,Z 186,A 108.7277,B 2.981,C 0.0301,E1 2.935,E2 344.8024} C_DIS
LIN {X -45.1292,Y 129.8002,Z 186,A 110.1289,B 2.981,C 0.0312,E1 2.9313,E2 343.401} C_DIS
LIN {X -48.3806,Y 128.6237,Z 186,A 111.6335,B 2.981,C 0.0321,E1 2.9273,E2 341.8897} C_DIS
LIN {X -52.9453,Y 126.8128,Z 186,A 113.7024,B 2.981,C 0.0339,E1 2.9219,E2 339.8195} C_DIS
LIN {X -56.2696,Y 125.3732,Z 186,A 115.1979,B 2.9809,C 0.0356,E1 2.9181,E2 338.3267} C_DIS
LIN {X -59.1547,Y 124.0379,Z 186,A 117.2645,B 2.9809,C 0.0332,E1 2.9127,E2 336.1702} C_DIS
LIN {X -63.9936,Y 121.6121,Z 186,A 118.5845,B 2.9809,C 0.0407,E1 2.9097,E2 334.9664} C_DIS
LIN {X -66.7769,Y 120.1089,Z 186,A 120.2771,B 2.9809,C 0.0405,E1 2.9054,E2 333.2294} C_DIS
LIN {X -71.56,Y 117.3223,Z 186,A 122.4775,B 2.9808,C 0.0441,E1 2.9002,E2 331.0437} C_DIS
LIN {X -74.508,Y 115.4727,Z 186,A 124.1456,B 2.9808,C 0.0451,E1 2.8962,E2 329.3501} C_DIS
LIN {X -78.1236,Y 113.058,Z 186,A 126.0359,B 2.9808,C 0.0474,E1 2.8918,E2 327.4516} C_DIS
LIN {X -81.7735,Y 110.4467,Z 186,A 127.9255,B 2.9807,C 0.0503,E1 2.8875,E2 325.5611} C_DIS
LIN {X -85.8941,Y 107.2734,Z 186,A 130.1262,B 2.9807,C 0.0538,E1 2.8826,E2 323.358} C_DIS
LIN {X -89.0632,Y 104.6565,Z 186,A 131.9164,B 2.9806,C 0.0564,E1 2.8788,E2 321.5596} C_DIS
LIN {X -92.5044,Y 101.6278,Z 186,A 133.9059,B 2.9806,C 0.0595,E1 2.8746,E2 319.5619} C_DIS
LIN {X -95.6679,Y 98.6555,Z 186,A 135.7924,B 2.9804,C 0.0626,E1 2.8708,E2 317.6672} C_DIS
LIN {X -98.6427,Y 95.6811,Z 186,A 137.607,B 2.9804,C 0.0657,E1 2.8672,E2 315.8465} C_DIS
LIN {X -101.5277,Y 92.6147,Z 186,A 139.4456,B 2.9804,C 0.0689,E1 2.8637,E2 313.999} C_DIS
LIN {X -104.577,Y 89.1567,Z 186,A 141.6061,B 2.9802,C 0.0719,E1 2.8597,E2 311.8104} C_DIS
LIN {X -106.6627,Y 86.6514,Z 186,A 142.8131,B 2.9802,C 0.0755,E1 2.8576,E2 310.6234} C_DIS
LIN {X -109.3742,Y 83.2024,Z 186,A 144.7143,B 2.98,C 0.0792,E1 2.8544,E2 308.7146} C_DIS
LIN {X -112.0382,Y 79.5792,Z 186,A 146.6315,B 2.98,C 0.0832,E1 2.8512,E2 306.7936} C_DIS
LIN {X -114.5775,Y 75.8772,Z 186,A 148.5921,B 2.9798,C 0.0872,E1 2.8482,E2 304.8234} C_DIS
LIN {X -116.3738,Y 73.0922,Z 186,A 150.0486,B 2.9798,C 0.0901,E1 2.846,E2 303.3587} C_DIS
LIN {X -118.6871,Y 69.273,Z 186,A 152.0208,B 2.9796,C 0.0942,E1 2.8431,E2 301.3742} C_DIS
LIN {X -120.8606,Y 65.4074,Z 186,A 153.9533,B 2.9795,C 0.0984,E1 2.8405,E2 299.4327} C_DIS
LIN {X -122.5905,Y 62.0993,Z 186,A 155.477,B 2.9793,C 0.1023,E1 2.8386,E2 297.9141} C_DIS
LIN {X -124.3658,Y 58.4685,Z 186,A 158.4415,B 2.9793,C 0.1019,E1 2.8349,E2 294.7898} C_DIS
LIN {X -127.5115,Y 51.2399,Z 186,A 160.6931,B 2.9789,C 0.1142,E1 2.8326,E2 292.6716} C_DIS
LIN {X -128.8963,Y 47.6527,Z 186,A 162.3436,B 2.9788,C 0.1182,E1 2.831,E2 291.0165} C_DIS
LIN {X -130.011,Y 44.5209,Z 186,A 163.7711,B 2.9786,C 0.1217,E1 2.8297,E2 289.5847} C_DIS
LIN {X -131.0312,Y 41.4212,Z 186,A 165.2908,B 2.9785,C 0.1248,E1 2.8284,E2 288.0461} C_DIS
LIN {X -131.9312,Y 38.4568,Z 186,A 166.6263,B 2.9783,C 0.1281,E1 2.8273,E2 286.706} C_DIS
LIN {X -132.8649,Y 35.0964,Z 186,A 168.1003,B 2.9782,C 0.132,E1 2.8262,E2 285.2306} C_DIS
LIN {X -133.8128,Y 31.2951,Z 186,A 169.7572,B 2.978,C 0.1364,E1 2.8251,E2 283.5719} C_DIS
LIN {X -134.6196,Y 27.6111,Z 186,A 171.5138,B 2.9778,C 0.1401,E1 2.8241,E2 281.7931} C_DIS
LIN {X -135.2678,Y 24.2362,Z 186,A 172.9873,B 2.9776,C 0.1439,E1 2.8234,E2 280.3155} C_DIS
LIN {X -135.8226,Y 20.9051,Z 186,A 174.4982,B 2.9775,C 0.1475,E1 2.8227,E2 278.7926} C_DIS
LIN {X -136.4134,Y 16.6225,Z 186,A 176.3534,B 2.9772,C 0.1523,E1 2.822,E2 276.932} C_DIS
LIN {X -136.7987,Y 13.0734,Z 186,A 177.9186,B 2.977,C 0.1562,E1 2.8216,E2 275.358} C_DIS
LIN {X -137.1268,Y 9.0221,Z 186,A 179.7801,B 2.9768,C 0.1604,E1 2.8212,E2 273.4765} C_DIS
LIN {X -137.332,Y 4.9887,Z 186,A -178.461,B 2.9765,C 0.1649,E1 2.821,E2 271.7091} C_DIS
LIN {X -137.4228,Y 0.4878,Z 186,A -176.4744,B 2.9763,C 0.1698,E1 2.821,E2 269.7097} C_DIS
LIN {X -137.3722,Y -3.7046,Z 186,A -174.7248,B 2.976,C 0.1747,E1 2.821,E2 267.961} C_DIS
LIN {X -137.2184,Y -7.5035,Z 186,A -173.0713,B 2.9757,C 0.1789,E1 2.8212,E2 266.2998} C_DIS
LIN {X -136.9567,Y -11.3027,Z 186,A -171.3815,B 2.9755,C 0.183,E1 2.8216,E2 264.5978} C_DIS
LIN {X -136.6139,Y -14.8824,Z 186,A -169.8653,B 2.9752,C 0.1872,E1 2.822,E2 263.0803} C_DIS
LIN {X -136.2045,Y -18.256,Z 186,A -168.2204,B 2.975,C 0.1903,E1 2.8226,E2 261.407} C_DIS
LIN {X -135.573,Y -22.4667,Z 186,A -166.4317,B 2.9747,C 0.1952,E1 2.8234,E2 259.6176} C_DIS
LIN {X -134.9184,Y -26.1131,Z 186,A -164.8826,B 2.9744,C 0.1994,E1 2.8242,E2 258.0687} C_DIS
LIN {X -134.2995,Y -29.1276,Z 186,A -163.5048,B 2.9742,C 0.2026,E1 2.825,E2 256.6794} C_DIS
LIN {X -133.5221,Y -32.5068,Z 186,A -161.9637,B 2.974,C 0.2062,E1 2.826,E2 255.1267} C_DIS
LIN {X -132.4326,Y -36.6941,Z 186,A -160.0768,B 2.9736,C 0.2107,E1 2.8274,E2 253.23} C_DIS
LIN {X -131.4275,Y -40.1441,Z 186,A -158.1277,B 2.9735,C 0.2131,E1 2.829,E2 251.223} C_DIS
LIN {X -130.2651,Y -43.7704,Z 186,A -156.8724,B 2.9731,C 0.2185,E1 2.8301,E2 250.0118} C_DIS
LIN {X -129.3225,Y -46.4802,Z 186,A -155.4435,B 2.9729,C 0.2208,E1 2.8314,E2 248.5531} C_DIS
LIN {X -127.941,Y -50.1592,Z 186,A -153.9224,B 2.9726,C 0.2255,E1 2.8329,E2 247.0481} C_DIS
LIN {X -126.725,Y -53.1556,Z 186,A -152.4806,B 2.9723,C 0.2286,E1 2.8345,E2 245.5946} C_DIS
LIN {X -125.1805,Y -56.7005,Z 186,A -150.8191,B 2.972,C 0.2325,E1 2.8364,E2 243.9274} C_DIS
LIN {X -123.8645,Y -59.5177,Z 186,A -149.441,B 2.9718,C 0.2354,E1 2.838,E2 242.5391} C_DIS
LIN {X -122.2146,Y -62.8377,Z 186,A -147.7521,B 2.9715,C 0.2386,E1 2.8402,E2 240.832} C_DIS
LIN {X -120.2605,Y -66.503,Z 186,A -145.9368,B 2.9712,C 0.2425,E1 2.8426,E2 239.0065} C_DIS
LIN {X -117.9281,Y -70.5568,Z 186,A -143.8906,B 2.9709,C 0.2467,E1 2.8455,E2 236.9483} C_DIS
LIN {X -115.5023,Y -74.4623,Z 186,A -141.8957,B 2.9705,C 0.2508,E1 2.8485,E2 234.9438} C_DIS
LIN {X -113.047,Y -78.1395,Z 186,A -139.9878,B 2.9702,C 0.2547,E1 2.8515,E2 233.0279} C_DIS
LIN {X -110.517,Y -81.6785,Z 186,A -138.1309,B 2.9699,C 0.2585,E1 2.8546,E2 231.1658} C_DIS
LIN {X -107.8452,Y -85.1749,Z 186,A -136.1757,B 2.9696,C 0.262,E1 2.858,E2 229.195} C_DIS
LIN {X -104.9637,Y -88.7018,Z 186,A -134.1814,B 2.9693,C 0.2655,E1 2.8616,E2 227.1885} C_DIS
LIN {X -98.993,Y -95.3193,Z 186,A -129.982,B 2.9688,C 0.2706,E1 2.8697,E2 222.9256} C_DIS
LIN {X -95.9845,Y -98.3479,Z 186,A -128.509,B 2.9684,C 0.2754,E1 2.8725,E2 221.4937} C_DIS
LIN {X -92.6925,Y -101.4569,Z 186,A -126.565,B 2.9681,C 0.2785,E1 2.8765,E2 219.5425} C_DIS
LIN {X -89.2906,Y -104.4632,Z 186,A -124.5978,B 2.9678,C 0.2814,E1 2.8807,E2 217.5655} C_DIS
LIN {X -85.7343,Y -107.4006,Z 186,A -122.6384,B 2.9675,C 0.2844,E1 2.8849,E2 215.6014} C_DIS
LIN {X -82.0168,Y -110.2655,Z 186,A -120.6756,B 2.9672,C 0.2875,E1 2.8893,E2 213.6378} C_DIS
LIN {X -78.4803,Y -112.8099,Z 186,A -118.8028,B 2.967,C 0.2899,E1 2.8936,E2 211.7575} C_DIS
LIN {X -74.8132,Y -115.2745,Z 186,A -116.9041,B 2.9668,C 0.2923,E1 2.8981,E2 209.8512} C_DIS
LIN {X -70.9584,Y -117.6867,Z 186,A -114.9569,B 2.9665,C 0.2945,E1 2.9027,E2 207.8971} C_DIS
LIN {X -67.4321,Y -119.742,Z 186,A -113.2107,B 2.9663,C 0.2964,E1 2.907,E2 206.1447} C_DIS
LIN {X -63.2585,Y -121.9981,Z 186,A -111.3007,B 2.9661,C 0.2991,E1 2.9117,E2 204.2436} C_DIS
LIN {X -60.5609,Y -123.3577,Z 186,A -109.9906,B 2.966,C 0.3002,E1 2.915,E2 202.9266} C_DIS
LIN {X -57.5502,Y -124.7905,Z 186,A -108.6029,B 2.9658,C 0.3017,E1 2.9185,E2 201.539} C_DIS
LIN {X -54.61,Y -126.1049,Z 186,A -107.226,B 2.9657,C 0.3028,E1 2.922,E2 200.1573} C_DIS
LIN {X -51.1719,Y -127.5389,Z 186,A -105.6574,B 2.9656,C 0.3041,E1 2.9261,E2 198.5863} C_DIS
LIN {X -47.9784,Y -128.7744,Z 186,A -104.1863,B 2.9655,C 0.3051,E1 2.9299,E2 197.1091} C_DIS
LIN {X -44.7292,Y -129.9388,Z 186,A -102.76,B 2.9653,C 0.3063,E1 2.9337,E2 195.6842} C_DIS
LIN {X -41.6245,Y -130.9662,Z 186,A -101.3641,B 2.9653,C 0.307,E1 2.9374,E2 194.2836} C_DIS
LIN {X -38.5246,Y -131.9113,Z 186,A -99.9958,B 2.9652,C 0.3078,E1 2.9411,E2 192.9126} C_DIS
LIN {X -35.1952,Y -132.8386,Z 186,A -98.491,B 2.9652,C 0.3082,E1 2.9452,E2 191.3988} C_DIS
LIN {X -31.7151,Y -133.7129,Z 186,A -97.0723,B 2.965,C 0.3094,E1 2.949,E2 189.9902} C_DIS
LIN {X -29.1327,Y -134.2984,Z 186,A -95.879,B 2.965,C 0.3094,E1 2.9523,E2 188.7844} C_DIS
LIN {X -25.5984,Y -135.0168,Z 186,A -94.3724,B 2.965,C 0.3099,E1 2.9564,E2 187.277} C_DIS
LIN {X -19.8623,Y -135.9796,Z 186,A -92.1269,B 2.9648,C 0.3118,E1 2.9626,E2 185.0548} C_DIS
LIN {X -15.6762,Y -136.5262,Z 186,A -90.2329,B 2.9648,C 0.3112,E1 2.9679,E2 183.1421} C_DIS
LIN {X -11.9695,Y -136.9003,Z 186,A -88.3201,B 2.9651,C 0.3088,E1 2.9733,E2 181.1801} C_DIS
LIN {X -8.5313,Y -137.157,Z 186,A -87.057,B 2.9649,C 0.3101,E1 2.9768,E2 179.9399} C_DIS
LIN {X -3.9502,Y -137.3654,Z 186,A -85.2549,B 2.9649,C 0.3107,E1 2.9818,E2 178.1519} C_DIS
LIN {X 0.1687,Y -137.4233,Z 186,A -83.4943,B 2.9649,C 0.3101,E1 2.9867,E2 176.3847} C_DIS
LIN {X 0.1687,Y -137.4233,Z 186,A -83.4943,B 2.9649,C 0.3101,E1 2.9867,E2 176.3847} C_DIS
Enddeposition()
LIN {X 0.9937,Y -138.3169,Z 186,A -83.3165,B 2.9402,C 0.3119,E1 2.9626,E2 176.2662} C_DIS
Startdeposition()
$VEL.CP = VEL_PRINT
LIN {X -2.527,Y -138.2991,Z 186,A -85.2918,B 2.9398,C 0.3158,E1 2.9569,E2 178.3122} C_DIS
LIN {X -6.1665,Y -138.1866,Z 186,A -86.7489,B 2.9398,C 0.3155,E1 2.9528,E2 179.7631} C_DIS
LIN {X -10.8553,Y -137.8975,Z 186,A -88.6985,B 2.9398,C 0.3155,E1 2.9474,E2 181.7141} C_DIS
LIN {X -15.0318,Y -137.5028,Z 186,A -90.4973,B 2.9398,C 0.3158,E1 2.9424,E2 183.5217} C_DIS
LIN {X -19.8019,Y -136.8972,Z 186,A -92.4455,B 2.9398,C 0.3151,E1 2.937,E2 185.4647} C_DIS
LIN {X -22.9999,Y -136.3964,Z 186,A -93.7951,B 2.9398,C 0.3148,E1 2.9332,E2 186.8161} C_DIS
LIN {X -26.2243,Y -135.8133,Z 186,A -95.2156,B 2.9398,C 0.3148,E1 2.9293,E2 188.2455} C_DIS
LIN {X -29.996,Y -135.0326,Z 186,A -96.7716,B 2.94,C 0.3138,E1 2.9251,E2 189.7968} C_DIS
LIN {X -33.2206,Y -134.2757,Z 186,A -98.1575,B 2.94,C 0.3132,E1 2.9213,E2 191.1851} C_DIS
LIN {X -36.155,Y -133.5139,Z 186,A -99.4145,B 2.9401,C 0.3125,E1 2.9179,E2 192.4425} C_DIS
LIN {X -39.5889,Y -132.5373,Z 186,A -100.924,B 2.9402,C 0.3118,E1 2.9138,E2 193.9566} C_DIS
LIN {X -42.8966,Y -131.5045,Z 186,A -102.3784,B 2.9402,C 0.3109,E1 2.9099,E2 195.4139} C_DIS
LIN {X -46.1125,Y -130.4117,Z 186,A -103.8056,B 2.9404,C 0.31,E1 2.9062,E2 196.8442} C_DIS
LIN {X -49.078,Y -129.3234,Z 186,A -105.1397,B 2.9404,C 0.309,E1 2.9027,E2 198.1819} C_DIS
LIN {X -52.5107,Y -127.9695,Z 186,A -106.689,B 2.9406,C 0.3078,E1 2.8986,E2 199.7344} C_DIS
LIN {X -55.6866,Y -126.6198,Z 186,A -108.144,B 2.9407,C 0.3066,E1 2.8949,E2 201.193} C_DIS
LIN {X -58.511,Y -125.3377,Z 186,A -109.4772,B 2.9409,C 0.3055,E1 2.8915,E2 202.5328} C_DIS
LIN {X -61.975,Y -123.6635,Z 186,A -111.079,B 2.941,C 0.3038,E1 2.8875,E2 204.136} C_DIS
LIN {X -65.0809,Y -122.0575,Z 186,A -112.6298,B 2.9411,C 0.3027,E1 2.8836,E2 205.7007} C_DIS
LIN {X -68.9205,Y -119.9313,Z 186,A -114.5251,B 2.9413,C 0.3009,E1 2.879,E2 207.6064} C_DIS
LIN {X -72.7065,Y -117.6747,Z 186,A -116.4085,B 2.9416,C 0.2988,E1 2.8744,E2 209.4976} C_DIS
LIN {X -76.3602,Y -115.3369,Z 186,A -118.2139,B 2.9418,C 0.2963,E1 2.8702,E2 211.3042} C_DIS
LIN {X -80.0917,Y -112.7781,Z 186,A -120.1764,B 2.942,C 0.294,E1 2.8657,E2 213.2784} C_DIS
LIN {X -83.6781,Y -110.1433,Z 186,A -122.0242,B 2.9423,C 0.2911,E1 2.8615,E2 215.1268} C_DIS
LIN {X -87.1051,Y -107.4532,Z 186,A -123.8939,B 2.9426,C 0.2885,E1 2.8574,E2 217.0051} C_DIS
LIN {X -90.5743,Y -104.5458,Z 186,A -125.8339,B 2.9429,C 0.2856,E1 2.8533,E2 218.9535} C_DIS
LIN {X -93.9394,Y -101.533,Z 186,A -127.7457,B 2.9432,C 0.2824,E1 2.8493,E2 220.8706} C_DIS
LIN {X -96.9492,Y -98.6623,Z 186,A -129.4928,B 2.9435,C 0.2793,E1 2.8458,E2 222.6206} C_DIS
LIN {X -99.9681,Y -95.602,Z 186,A -131.3681,B 2.9437,C 0.2764,E1 2.8421,E2 224.5082} C_DIS
LIN {X -102.9505,Y -92.3827,Z 186,A -133.223,B 2.9441,C 0.2729,E1 2.8386,E2 226.3677} C_DIS
LIN {X -105.6792,Y -89.2494,Z 186,A -135.0335,B 2.9443,C 0.2698,E1 2.8353,E2 228.1897} C_DIS
LIN {X -108.5045,Y -85.7924,Z 186,A -137.0005,B 2.9447,C 0.2664,E1 2.8318,E2 230.1717} C_DIS
LIN {X -111.2118,Y -82.2526,Z 186,A -138.8372,B 2.945,C 0.2623,E1 2.8288,E2 232.0068} C_DIS
LIN {X -113.7436,Y -78.7139,Z 186,A -140.7539,B 2.9453,C 0.2588,E1 2.8256,E2 233.9379} C_DIS
LIN {X -116.2588,Y -74.9496,Z 186,A -142.719,B 2.9457,C 0.2549,E1 2.8226,E2 235.9143} C_DIS
LIN {X -118.5453,Y -71.2776,Z 186,A -144.5708,B 2.946,C 0.2509,E1 2.8199,E2 237.7733} C_DIS
LIN {X -120.7976,Y -67.3907,Z 186,A -146.4997,B 2.9464,C 0.2467,E1 2.8172,E2 239.7105} C_DIS
LIN {X -122.8711,Y -63.5315,Z 186,A -148.3168,B 2.9467,C 0.2423,E1 2.8149,E2 241.5272} C_DIS
LIN {X -124.2418,Y -60.8027,Z 186,A -149.6705,B 2.947,C 0.2395,E1 2.8132,E2 242.892} C_DIS
LIN {X -125.9128,Y -57.2672,Z 186,A -151.3289,B 2.9473,C 0.2356,E1 2.8112,E2 244.5548} C_DIS
LIN {X -127.3053,Y -54.101,Z 186,A -152.8261,B 2.9475,C 0.2322,E1 2.8095,E2 246.0598} C_DIS
LIN {X -128.6121,Y -50.9164,Z 186,A -154.3168,B 2.9478,C 0.2288,E1 2.808,E2 247.5584} C_DIS
LIN {X -129.8332,Y -47.7168,Z 186,A -155.801,B 2.9481,C 0.2253,E1 2.8065,E2 249.0504} C_DIS
LIN {X -130.9688,Y -44.5056,Z 186,A -157.2773,B 2.9483,C 0.2219,E1 2.8052,E2 250.5345} C_DIS
LIN {X -131.8374,Y -41.8547,Z 186,A -158.4842,B 2.9486,C 0.219,E1 2.8041,E2 251.7475} C_DIS
LIN {X -132.8146,Y -38.6418,Z 186,A -159.9446,B 2.9488,C 0.2155,E1 2.8029,E2 253.2161} C_DIS
LIN {X -133.7142,Y -35.4038,Z 186,A -161.401,B 2.9491,C 0.212,E1 2.8019,E2 254.6802} C_DIS
LIN {X -134.5272,Y -32.1773,Z 186,A -162.8453,B 2.9493,C 0.2085,E1 2.8009,E2 256.1322} C_DIS
LIN {X -135.3167,Y -28.6802,Z 186,A -164.4201,B 2.9496,C 0.2047,E1 2.8,E2 257.7178} C_DIS
LIN {X -136.0148,Y -25.1699,Z 186,A -165.9565,B 2.9498,C 0.2009,E1 2.7991,E2 259.2604} C_DIS
LIN {X -136.5692,Y -21.9638,Z 186,A -167.3698,B 2.9501,C 0.1974,E1 2.7985,E2 260.6813} C_DIS
LIN {X -137.1677,Y -17.8312,Z 186,A -169.1971,B 2.9504,C 0.1929,E1 2.7978,E2 262.5201} C_DIS
LIN {X -137.613,Y -14.0076,Z 186,A -170.8564,B 2.9507,C 0.1887,E1 2.7973,E2 264.1869} C_DIS
LIN {X -137.9716,Y -9.8407,Z 186,A -172.7295,B 2.9509,C 0.1843,E1 2.7968,E2 266.0768} C_DIS
LIN {X -138.1866,Y -6.1665,Z 186,A -174.2735,B 2.9512,C 0.1801,E1 2.7966,E2 267.6225} C_DIS
LIN {X -138.3156,Y -1.5317,Z 186,A -176.224,B 2.9515,C 0.1748,E1 2.7965,E2 269.5755} C_DIS
LIN {X -138.3156,Y 1.5317,Z 186,A -177.6236,B 2.9517,C 0.1716,E1 2.7965,E2 270.9909} C_DIS
LIN {X -138.2471,Y 4.6152,Z 186,A -178.9693,B 2.9519,C 0.1683,E1 2.7966,E2 272.3445} C_DIS
LIN {X -138.0665,Y 8.4024,Z 186,A 179.3395,B 2.9521,C 0.1643,E1 2.7969,E2 274.0499} C_DIS
LIN {X -137.8208,Y 11.7631,Z 186,A 177.8886,B 2.9523,C 0.1605,E1 2.7972,E2 275.5068} C_DIS
LIN {X -137.5028,Y 15.0318,Z 186,A 176.4163,B 2.9525,C 0.1571,E1 2.7976,E2 276.9924} C_DIS
LIN {X -136.8972,Y 19.8019,Z 186,A 174.3774,B 2.9528,C 0.1517,E1 2.7984,E2 279.0359} C_DIS
LIN {X -136.3964,Y 22.9999,Z 186,A 172.9074,B 2.9529,C 0.1484,E1 2.799,E2 280.5212} C_DIS
LIN {X -135.7077,Y 26.7767,Z 186,A 171.2932,B 2.9532,C 0.1441,E1 2.7999,E2 282.1374} C_DIS
LIN {X -135.0326,Y 29.996,Z 186,A 169.8602,B 2.9533,C 0.1406,E1 2.8007,E2 283.5783} C_DIS
LIN {X -134.4038,Y 32.6891,Z 186,A 168.6514,B 2.9535,C 0.1377,E1 2.8015,E2 284.7941} C_DIS
LIN {X -133.5668,Y 35.9568,Z 186,A 167.1407,B 2.9536,C 0.1343,E1 2.8026,E2 286.318} C_DIS
LIN {X -132.5124,Y 39.6739,Z 186,A 165.5056,B 2.9538,C 0.1301,E1 2.8039,E2 287.9564} C_DIS
LIN {X -131.5045,Y 42.8966,Z 186,A 164.0372,B 2.954,C 0.1266,E1 2.8051,E2 289.4324} C_DIS
LIN {X -130.4117,Y 46.1125,Z 186,A 162.5607,B 2.9541,C 0.1231,E1 2.8065,E2 290.9165} C_DIS
LIN {X -129.4308,Y 48.7913,Z 186,A 161.3131,B 2.9542,C 0.1202,E1 2.8077,E2 292.1715} C_DIS
LIN {X -127.9695,Y 52.5107,Z 186,A 159.5853,B 2.9544,C 0.1162,E1 2.8095,E2 293.9072} C_DIS
LIN {X -126.6198,Y 55.6866,Z 186,A 158.0877,B 2.9545,C 0.1127,E1 2.8112,E2 295.4122} C_DIS
LIN {X -125.1844,Y 58.8425,Z 186,A 156.5839,B 2.9547,C 0.1093,E1 2.8129,E2 296.9233} C_DIS
LIN {X -123.8259,Y 61.6458,Z 186,A 155.2087,B 2.9547,C 0.1064,E1 2.8146,E2 298.308} C_DIS
LIN {X -122.0575,Y 65.0809,Z 186,A 153.5964,B 2.9549,C 0.1025,E1 2.8167,E2 299.9205} C_DIS
LIN {X -120.3671,Y 68.1567,Z 186,A 151.9205,B 2.9549,C 0.0998,E1 2.819,E2 301.6229} C_DIS
LIN {X -118.1364,Y 71.9539,Z 186,A 150.0115,B 2.9551,C 0.0957,E1 2.8218,E2 303.5409} C_DIS
LIN {X -115.7767,Y 75.6923,Z 186,A 148.1014,B 2.9552,C 0.0917,E1 2.8247,E2 305.4594} C_DIS
LIN {X -113.2903,Y 79.3654,Z 186,A 146.2353,B 2.9554,C 0.0877,E1 2.8277,E2 307.3276} C_DIS
LIN {X -110.68,Y 82.9669,Z 186,A 144.318,B 2.9554,C 0.0838,E1 2.8308,E2 309.2528} C_DIS
LIN {X -107.9488,Y 86.4906,Z 186,A 142.3983,B 2.9556,C 0.0801,E1 2.8342,E2 311.18} C_DIS
LIN {X -105.3048,Y 89.6899,Z 186,A 140.6466,B 2.9556,C 0.0766,E1 2.8373,E2 312.9344} C_DIS
LIN {X -102.7398,Y 92.618,Z 186,A 138.905,B 2.9558,C 0.0739,E1 2.8406,E2 314.6906} C_DIS
LIN {X -99.6904,Y 95.8926,Z 186,A 137.0983,B 2.9558,C 0.07,E1 2.844,E2 316.4902} C_DIS
LIN {X -96.9663,Y 98.6454,Z 186,A 135.3831,B 2.9559,C 0.0673,E1 2.8475,E2 318.2178} C_DIS
LIN {X -94.1707,Y 101.3176,Z 186,A 133.7394,B 2.9559,C 0.0645,E1 2.8508,E2 319.8653} C_DIS
LIN {X -90.9605,Y 104.2092,Z 186,A 131.8636,B 2.956,C 0.0617,E1 2.8548,E2 321.7503} C_DIS
LIN {X -87.6327,Y 107.0228,Z 186,A 129.9802,B 2.956,C 0.0589,E1 2.8588,E2 323.642} C_DIS
LIN {X -83.9281,Y 109.9521,Z 186,A 128.0188,B 2.9561,C 0.0557,E1 2.8631,E2 325.6026} C_DIS
LIN {X -80.5595,Y 112.4435,Z 186,A 126.184,B 2.9561,C 0.0534,E1 2.8673,E2 327.4482} C_DIS
LIN {X -76.9094,Y 114.971,Z 186,A 124.2972,B 2.9562,C 0.0509,E1 2.8717,E2 329.3395} C_DIS
LIN {X -72.9714,Y 117.5098,Z 186,A 122.36,B 2.9562,C 0.0481,E1 2.8762,E2 331.2749} C_DIS
LIN {X -69.4132,Y 119.6461,Z 186,A 120.5694,B 2.9563,C 0.0462,E1 2.8806,E2 333.0731} C_DIS
LIN {X -65.5802,Y 121.7893,Z 186,A 118.6932,B 2.9563,C 0.0442,E1 2.8852,E2 334.955} C_DIS
LIN {X -61.975,Y 123.6635,Z 186,A 117.0691,B 2.9563,C 0.0419,E1 2.8892,E2 336.5709} C_DIS
LIN {X -58.8425,Y 125.1844,Z 186,A 115.5997,B 2.9563,C 0.0404,E1 2.8929,E2 338.0426} C_DIS
LIN {X -55.6866,Y 126.6198,Z 186,A 114.1387,B 2.9564,C 0.039,E1 2.8967,E2 339.5057} C_DIS
LIN {X -53.0723,Y 127.7349,Z 186,A 112.9426,B 2.9564,C 0.038,E1 2.8997,E2 340.7032} C_DIS
LIN {X -49.8826,Y 129.014,Z 186,A 111.4978,B 2.9564,C 0.0368,E1 2.9035,E2 342.1497} C_DIS
LIN {X -46.679,Y 130.2074,Z 186,A 110.0572,B 2.9564,C 0.0357,E1 2.9073,E2 343.5924} C_DIS
LIN {X -43.1331,Y 131.4258,Z 186,A 108.5087,B 2.9564,C 0.0345,E1 2.9114,E2 345.1395} C_DIS
LIN {X -39.6739,Y 132.5124,Z 186,A 106.9708,B 2.9564,C 0.0336,E1 2.9155,E2 346.6809} C_DIS
LIN {X -37.0173,Y 133.2766,Z 186,A 105.821,B 2.9564,C 0.0329,E1 2.9186,E2 347.8305} C_DIS
LIN {X -33.8254,Y 134.1222,Z 186,A 104.4097,B 2.9564,C 0.0323,E1 2.9224,E2 349.2463} C_DIS
LIN {X -29.996,Y 135.0326,Z 186,A 102.7925,B 2.9565,C 0.0314,E1 2.9268,E2 350.8611} C_DIS
LIN {X -26.7767,Y 135.7077,Z 186,A 101.4214,B 2.9565,C 0.0309,E1 2.9306,E2 352.2325} C_DIS
LIN {X -23.5655,Y 136.302,Z 186,A 100.0624,B 2.9565,C 0.0304,E1 2.9343,E2 353.5915} C_DIS
LIN {X -20.3652,Y 136.8167,Z 186,A 98.7149,B 2.9565,C 0.03,E1 2.9381,E2 354.9389} C_DIS
LIN {X -17.1784,Y 137.2533,Z 186,A 97.3793,B 2.9565,C 0.0297,E1 2.9418,E2 356.2743} C_DIS
LIN {X -14.0076,Y 137.613,Z 186,A 96.0559,B 2.9565,C 0.0295,E1 2.9454,E2 357.5973} C_DIS
LIN {X -10.8553,Y 137.8975,Z 186,A 94.7449,B 2.9565,C 0.0294,E1 2.9491,E2 358.9076} C_DIS
LIN {X -7.7238,Y 138.1083,Z 186,A 93.4463,B 2.9565,C 0.0294,E1 2.9527,E2 360.2055} C_DIS
LIN {X -3.6963,Y 138.2727,Z 186,A 91.7145,B 2.9565,C 0.0297,E1 2.9576,E2 361.9439} C_DIS
LIN {X 0,Y 138.3241,Z 186,A 90.2543,B 2.9565,C 0.0295,E1 2.9616,E2 363.395} C_DIS
LIN {X 4.6152,Y 138.2471,Z 186,A 88.3444,B 2.9565,C 0.0298,E1 2.967,E2 365.3038} C_DIS
LIN {X 8.6969,Y 138.0484,Z 186,A 86.6864,B 2.9565,C 0.03,E1 2.9716,E2 366.957} C_DIS
LIN {X 11.743,Y 137.8225,Z 186,A 85.3764,B 2.9565,C 0.0308,E1 2.9753,E2 368.2718} C_DIS
LIN {X 15.0318,Y 137.5028,Z 186,A 83.9807,B 2.9565,C 0.0315,E1 2.9791,E2 369.6704} C_DIS
LIN {X 19.8019,Y 136.8972,Z 186,A 82.0562,B 2.9565,C 0.0321,E1 2.9845,E2 371.5861} C_DIS
LIN {X 22.9999,Y 136.3964,Z 186,A 80.6715,B 2.9565,C 0.0332,E1 2.9883,E2 372.9756} C_DIS
LIN {X 26.7767,Y 135.7077,Z 186,A 79.1516,B 2.9565,C 0.0337,E1 2.9924,E2 374.4867} C_DIS
LIN {X 29.996,Y 135.0326,Z 186,A 77.8036,B 2.9565,C 0.0346,E1 2.9961,E2 375.8325} C_DIS
LIN {X 32.9749,Y 134.3349,Z 186,A 76.5658,B 2.9565,C 0.0353,E1 2.9995,E2 377.0664} C_DIS
LIN {X 36.0096,Y 133.5527,Z 186,A 75.2433,B 2.9565,C 0.0366,E1 3.0031,E2 378.3914} C_DIS
LIN {X 39.6739,Y 132.5124,Z 186,A 73.7137,B 2.9565,C 0.0377,E1 3.0071,E2 379.9149} C_DIS
LIN {X 42.8966,Y 131.5045,Z 186,A 72.3364,B 2.9565,C 0.0389,E1 3.0108,E2 381.2893} C_DIS
LIN {X 45.8895,Y 130.489,Z 186,A 71.0438,B 2.9565,C 0.0401,E1 3.0142,E2 382.5795} C_DIS
LIN {X 49.3183,Y 129.2334,Z 186,A 69.5621,B 2.9564,C 0.0415,E1 3.0181,E2 384.0573} C_DIS
LIN {X 52.5107,Y 127.9695,Z 186,A 68.1662,B 2.9564,C 0.043,E1 3.0217,E2 385.4498} C_DIS
LIN {X 55.2493,Y 126.8088,Z 186,A 66.9208,B 2.9564,C 0.0446,E1 3.0249,E2 386.6966} C_DIS
LIN {X 58.8425,Y 125.1844,Z 186,A 65.3585,B 2.9564,C 0.0461,E1 3.0288,E2 388.2501} C_DIS
LIN {X 61.975,Y 123.6635,Z 186,A 63.9474,B 2.9563,C 0.0478,E1 3.0324,E2 389.6572} C_DIS
LIN {X 65.5802,Y 121.7893,Z 186,A 62.2626,B 2.9563,C 0.0502,E1 3.0365,E2 391.342} C_DIS
LIN {X 69.4132,Y 119.6461,Z 186,A 60.4874,B 2.9563,C 0.0526,E1 3.0408,E2 393.1118} C_DIS
LIN {X 72.9714,Y 117.5098,Z 186,A 58.7635,B 2.9562,C 0.0553,E1 3.045,E2 394.8362} C_DIS
LIN {X 76.9094,Y 114.971,Z 186,A 56.9226,B 2.9562,C 0.0576,E1 3.0492,E2 396.6648} C_DIS
LIN {X 80.5595,Y 112.4435,Z 186,A 55.1479,B 2.9561,C 0.0602,E1 3.0533,E2 398.4316} C_DIS
LIN {X 83.9281,Y 109.9521,Z 186,A 53.4013,B 2.956,C 0.0634,E1 3.0572,E2 400.1796} C_DIS
LIN {X 87.6327,Y 107.0228,Z 186,A 51.5578,B 2.956,C 0.066,E1 3.0612,E2 402.0094} C_DIS
LIN {X 90.8457,Y 104.3093,Z 186,A 49.8593,B 2.9559,C 0.069,E1 3.0648,E2 403.7027} C_DIS
LIN {X 93.9394,Y 101.533,Z 186,A 48.2401,B 2.9559,C 0.0715,E1 3.0681,E2 405.3094} C_DIS
LIN {X 96.9392,Y 98.672,Z 186,A 46.523,B 2.9557,C 0.075,E1 3.0715,E2 407.0267} C_DIS
LIN {X 100.0905,Y 95.474,Z 186,A 44.7849,B 2.9557,C 0.0778,E1 3.0749,E2 408.7501} C_DIS
LIN {X 102.7398,Y 92.618,Z 186,A 43.1514,B 2.9556,C 0.0814,E1 3.078,E2 410.3864} C_DIS
LIN {X 105.6792,Y 89.2494,Z 186,A 41.4439,B 2.9555,C 0.0842,E1 3.0811,E2 412.0763} C_DIS
LIN {X 108.145,Y 86.244,Z 186,A 39.8085,B 2.9554,C 0.088,E1 3.0839,E2 413.7151} C_DIS
LIN {X 110.8652,Y 82.7182,Z 186,A 38.0303,B 2.9553,C 0.0916,E1 3.0869,E2 415.4856} C_DIS
LIN {X 113.6184,Y 78.8938,Z 186,A 36.2032,B 2.9551,C 0.095,E1 3.0899,E2 417.2976} C_DIS
LIN {X 115.9469,Y 75.4301,Z 186,A 34.496,B 2.9551,C 0.099,E1 3.0925,E2 419.0027} C_DIS
LIN {X 118.4317,Y 71.4655,Z 186,A 32.6841,B 2.9549,C 0.1025,E1 3.0951,E2 420.7994} C_DIS
LIN {X 120.5191,Y 67.8862,Z 186,A 30.9921,B 2.9548,C 0.1065,E1 3.0975,E2 422.4889} C_DIS
LIN {X 122.6674,Y 63.9195,Z 186,A 29.2577,B 2.9546,C 0.11,E1 3.0997,E2 424.2071} C_DIS
LIN {X 124.4346,Y 60.4119,Z 186,A 27.7309,B 2.9546,C 0.1132,E1 3.1016,E2 425.722} C_DIS
LIN {X 125.9128,Y 57.2672,Z 186,A 26.3538,B 2.9544,C 0.1163,E1 3.1032,E2 427.0918} C_DIS
LIN {X 127.0579,Y 54.6732,Z 186,A 25.2292,B 2.9543,C 0.1189,E1 3.1045,E2 428.2106} C_DIS
LIN {X 128.3852,Y 51.4794,Z 186,A 23.8614,B 2.9542,C 0.122,E1 3.1059,E2 429.5709} C_DIS
LIN {X 129.6214,Y 48.2823,Z 186,A 22.5045,B 2.954,C 0.1252,E1 3.1072,E2 430.9204} C_DIS
LIN {X 130.7876,Y 45.0282,Z 186,A 21.1136,B 2.9539,C 0.1286,E1 3.1085,E2 432.3068} C_DIS
LIN {X 131.943,Y 41.5239,Z 186,A 19.6665,B 2.9537,C 0.132,E1 3.1097,E2 433.7443} C_DIS
LIN {X 132.9847,Y 38.061,Z 186,A 18.248,B 2.9536,C 0.1353,E1 3.1109,E2 435.1536} C_DIS
LIN {X 133.7042,Y 35.4414,Z 186,A 17.17,B 2.9535,C 0.1379,E1 3.1116,E2 436.2261} C_DIS
LIN {X 134.5614,Y 32.0352,Z 186,A 15.7549,B 2.9533,C 0.1415,E1 3.1126,E2 437.6368} C_DIS
LIN {X 135.3803,Y 28.3855,Z 186,A 14.3095,B 2.9531,C 0.1448,E1 3.1134,E2 439.0699} C_DIS
LIN {X 136.0148,Y 25.1699,Z 186,A 13.0155,B 2.953,C 0.1479,E1 3.1141,E2 440.3566} C_DIS
LIN {X 136.5692,Y 21.9638,Z 186,A 11.731,B 2.9528,C 0.1511,E1 3.1147,E2 441.6337} C_DIS
LIN {X 137.0447,Y 18.7699,Z 186,A 10.4567,B 2.9527,C 0.1542,E1 3.1152,E2 442.9008} C_DIS
LIN {X 137.3758,Y 16.1515,Z 186,A 9.3646,B 2.9525,C 0.1572,E1 3.1156,E2 443.9933} C_DIS
LIN {X 137.7241,Y 12.8508,Z 186,A 8.0749,B 2.9523,C 0.1602,E1 3.1159,E2 445.2729} C_DIS
LIN {X 137.9716,Y 9.8407,Z 186,A 6.8644,B 2.9522,C 0.1634,E1 3.1162,E2 446.479} C_DIS
LIN {X 138.2193,Y 5.3287,Z 186,A 5.1086,B 2.9519,C 0.1675,E1 3.1164,E2 448.221} C_DIS
LIN {X 138.3156,Y 1.5317,Z 186,A 3.6916,B 2.9518,C 0.1704,E1 3.1164,E2 449.619} C_DIS
LIN {X 138.3156,Y -1.5317,Z 186,A 2.4222,B 2.9516,C 0.174,E1 3.1164,E2 450.8893} C_DIS
LIN {X 138.2471,Y -4.6152,Z 186,A 1.201,B 2.9514,C 0.177,E1 3.1164,E2 452.1041} C_DIS
LIN {X 138.0819,Y -8.1525,Z 186,A -0.2566,B 2.9511,C 0.1811,E1 3.1162,E2 453.5614} C_DIS
LIN {X 137.8263,Y -11.6987,Z 186,A -1.6351,B 2.9509,C 0.1843,E1 3.1159,E2 454.9287} C_DIS
LIN {X 137.5028,Y -15.0318,Z 186,A -2.9866,B 2.9507,C 0.1879,E1 3.1155,E2 456.2765} C_DIS
LIN {X 136.8972,Y -19.8019,Z 186,A -4.8394,B 2.9504,C 0.1921,E1 3.1148,E2 458.1128} C_DIS
LIN {X 136.3964,Y -22.9999,Z 186,A -6.1736,B 2.9502,C 0.1957,E1 3.1142,E2 459.4471} C_DIS
LIN {X 135.7077,Y -26.7767,Z 186,A -7.6414,B 2.95,C 0.199,E1 3.1134,E2 460.9002} C_DIS
LIN {X 135.0326,Y -29.996,Z 186,A -8.9443,B 2.9498,C 0.2022,E1 3.1127,E2 462.1964} C_DIS
LIN {X 134.2757,Y -33.2206,Z 186,A -10.2569,B 2.9495,C 0.2053,E1 3.1118,E2 463.5023} C_DIS
LIN {X 133.564,Y -35.9671,Z 186,A -11.3774,B 2.9494,C 0.208,E1 3.111,E2 464.6164} C_DIS
LIN {X 132.607,Y -39.351,Z 186,A -12.7947,B 2.9491,C 0.2116,E1 3.1099,E2 466.0297} C_DIS
LIN {X 131.5045,Y -42.8966,Z 186,A -14.2466,B 2.9489,C 0.2149,E1 3.1087,E2 467.4716} C_DIS
LIN {X 130.4117,Y -46.1125,Z 186,A -15.5933,B 2.9486,C 0.2181,E1 3.1075,E2 468.8116} C_DIS
LIN {X 129.2586,Y -49.2509,Z 186,A -16.9105,B 2.9484,C 0.2212,E1 3.1062,E2 470.1209} C_DIS
LIN {X 128.1125,Y -52.1559,Z 186,A -18.1834,B 2.9482,C 0.2244,E1 3.1049,E2 471.392} C_DIS
LIN {X 126.6198,Y -55.6866,Z 186,A -19.6802,B 2.9479,C 0.2277,E1 3.1032,E2 472.8783} C_DIS
LIN {X 125.3726,Y -58.4353,Z 186,A -20.8764,B 2.9477,C 0.2304,E1 3.1019,E2 474.0683} C_DIS
LIN {X 123.6635,Y -61.975,Z 186,A -22.4398,B 2.9474,C 0.2339,E1 3.0999,E2 475.6245} C_DIS
LIN {X 122.0575,Y -65.0809,Z 186,A -23.7963,B 2.9472,C 0.2367,E1 3.0982,E2 476.9701} C_DIS
LIN {X 120.3671,Y -68.1567,Z 186,A -25.3371,B 2.9468,C 0.2412,E1 3.0961,E2 478.5234} C_DIS
LIN {X 118.1364,Y -71.9539,Z 186,A -27.0891,B 2.9465,C 0.245,E1 3.0936,E2 480.2674} C_DIS
LIN {X 115.7767,Y -75.6923,Z 186,A -28.8488,B 2.9462,C 0.2488,E1 3.0909,E2 482.0192} C_DIS
LIN {X 113.3621,Y -79.2623,Z 186,A -30.5352,B 2.9459,C 0.2521,E1 3.0883,E2 483.694} C_DIS
LIN {X 110.68,Y -82.9669,Z 186,A -32.3443,B 2.9456,C 0.2557,E1 3.0853,E2 485.4933} C_DIS
LIN {X 107.9488,Y -86.4906,Z 186,A -34.1224,B 2.9453,C 0.2593,E1 3.0822,E2 487.2639} C_DIS
LIN {X 105.3048,Y -89.6899,Z 186,A -35.7272,B 2.945,C 0.262,E1 3.0794,E2 488.8549} C_DIS
LIN {X 102.7398,Y -92.618,Z 186,A -37.3582,B 2.9447,C 0.2657,E1 3.0763,E2 490.4896} C_DIS
LIN {X 99.6904,Y -95.8926,Z 186,A -39.0514,B 2.9445,C 0.2682,E1 3.0731,E2 492.163} C_DIS
LIN {X 96.9492,Y -98.6623,Z 186,A -40.6564,B 2.9442,C 0.2715,E1 3.07,E2 493.768} C_DIS
LIN {X 94.1707,Y -101.3176,Z 186,A -42.1889,B 2.9439,C 0.2742,E1 3.0669,E2 495.294} C_DIS
LIN {X 90.965,Y -104.2052,Z 186,A -43.9453,B 2.9436,C 0.2774,E1 3.0632,E2 497.0477} C_DIS
LIN {X 87.6327,Y -107.0228,Z 186,A -45.7156,B 2.9433,C 0.2805,E1 3.0594,E2 498.8144} C_DIS
LIN {X 83.9281,Y -109.9521,Z 186,A -47.5636,B 2.9431,C 0.2831,E1 3.0554,E2 500.6494} C_DIS
LIN {X 80.5595,Y -112.4435,Z 186,A -49.295,B 2.9428,C 0.2862,E1 3.0514,E2 502.3816} C_DIS
LIN {X 76.9094,Y -114.971,Z 186,A -51.0807,B 2.9425,C 0.2888,E1 3.0473,E2 504.1617} C_DIS
LIN {X 72.9714,Y -117.5098,Z 186,A -52.9197,B 2.9423,C 0.2911,E1 3.043,E2 505.9886} C_DIS
LIN {X 69.4132,Y -119.6461,Z 186,A -54.6402,B 2.9421,C 0.2938,E1 3.0389,E2 507.7105} C_DIS
LIN {X 65.6845,Y -121.7332,Z 186,A -56.3895,B 2.9418,C 0.2963,E1 3.0346,E2 509.4583} C_DIS
LIN {X 61.975,Y -123.6635,Z 186,A -57.967,B 2.9417,C 0.2974,E1 3.0307,E2 511.0164} C_DIS
LIN {X 58.8425,Y -125.1844,Z 186,A -59.3755,B 2.9415,C 0.2991,E1 3.0272,E2 512.4214} C_DIS
LIN {X 55.6866,Y -126.6198,Z 186,A -60.779,B 2.9414,C 0.3007,E1 3.0236,E2 513.8215} C_DIS
LIN {X 52.5107,Y -127.9695,Z 186,A -62.1774,B 2.9412,C 0.3022,E1 3.02,E2 515.2168} C_DIS
LIN {X 49.6328,Y -129.1111,Z 186,A -63.4527,B 2.9411,C 0.3036,E1 3.0167,E2 516.4918} C_DIS
LIN {X 46.1125,Y -130.4117,Z 186,A -64.9564,B 2.9409,C 0.3049,E1 3.0127,E2 517.9899} C_DIS
LIN {X 43.2407,Y -131.39,Z 186,A -66.198,B 2.9408,C 0.3061,E1 3.0094,E2 519.2303} C_DIS
LIN {X 39.6739,Y -132.5124,Z 186,A -67.7108,B 2.9407,C 0.3074,E1 3.0054,E2 520.7393} C_DIS
LIN {X 37.0173,Y -133.2766,Z 186,A -68.836,B 2.9406,C 0.3083,E1 3.0024,E2 521.8624} C_DIS
LIN {X 33.7903,Y -134.1311,Z 186,A -70.1966,B 2.9405,C 0.3093,E1 2.9987,E2 523.2209} C_DIS
LIN {X 30.4507,Y -134.9287,Z 186,A -71.6343,B 2.9403,C 0.3105,E1 2.9948,E2 524.6616} C_DIS
LIN {X 26.7767,Y -135.7077,Z 186,A -73.132,B 2.9403,C 0.3112,E1 2.9907,E2 526.1525} C_DIS
LIN {X 23.5655,Y -136.302,Z 186,A -74.4671,B 2.9402,C 0.312,E1 2.987,E2 527.486} C_DIS
LIN {X 20.3652,Y -136.8167,Z 186,A -75.7938,B 2.9402,C 0.3127,E1 2.9834,E2 528.8114} C_DIS
LIN {X 17.1784,Y -137.2533,Z 186,A -77.1118,B 2.94,C 0.3133,E1 2.9797,E2 530.1281} C_DIS
LIN {X 12.429,Y -137.7646,Z 186,A -79.0717,B 2.94,C 0.3141,E1 2.9743,E2 532.0866} C_DIS
LIN {X 9.8407,Y -137.9716,Z 186,A -80.19,B 2.9399,C 0.3148,E1 2.9711,E2 533.2112} C_DIS
LIN {X 6.1665,Y -138.1866,Z 186,A -81.6516,B 2.9399,C 0.3148,E1 2.9671,E2 534.6651} C_DIS
LIN {X 2.3383,Y -138.3022,Z 186,A -83.2503,B 2.9399,C 0.3153,E1 2.9626,E2 536.2662} C_DIS
LIN {X 2.3383,Y -138.3022,Z 186,A -83.2503,B 2.9399,C 0.3153,E1 2.9626,E2 536.2662} C_DIS
Enddeposition()
LIN {X 0.9954,Y -139.2169,Z 186,A -83.7103,B 2.9159,C 0.3153,E1 2.9375,E2 536.7509} C_DIS
Startdeposition()
$VEL.CP = VEL_PRINT
LIN {X 3.3698,Y -139.1819,Z 186,A -82.1633,B 2.9164,C 0.3111,E1 2.942,E2 535.1259} C_DIS
LIN {X 7.0907,Y -139.0411,Z 186,A -80.6528,B 2.9164,C 0.3108,E1 2.9462,E2 533.6175} C_DIS
LIN {X 10.7915,Y -138.8044,Z 186,A -79.0063,B 2.9166,C 0.3093,E1 2.9509,E2 531.9537} C_DIS
LIN {X 14.778,Y -138.4352,Z 186,A -77.5075,B 2.9166,C 0.3097,E1 2.955,E2 530.4745} C_DIS
LIN {X 21.655,Y -137.5276,Z 186,A -74.6596,B 2.9166,C 0.3082,E1 2.9629,E2 527.6259} C_DIS
LIN {X 27.9801,Y -136.3811,Z 186,A -72.0217,B 2.9169,C 0.3064,E1 2.9701,E2 524.9876} C_DIS
LIN {X 31.1093,Y -135.7013,Z 186,A -70.3539,B 2.9173,C 0.3026,E1 2.9748,E2 523.2709} C_DIS
LIN {X 35.0721,Y -134.7337,Z 186,A -69.0791,B 2.9171,C 0.3044,E1 2.9781,E2 522.0507} C_DIS
LIN {X 38.8739,Y -133.6843,Z 186,A -67.6026,B 2.9171,C 0.304,E1 2.982,E2 520.5932} C_DIS
LIN {X 42.1104,Y -132.7004,Z 186,A -66.1559,B 2.9173,C 0.3022,E1 2.9859,E2 519.138} C_DIS
LIN {X 45.3965,Y -131.6123,Z 186,A -64.7034,B 2.9175,C 0.3005,E1 2.9898,E2 517.6808} C_DIS
LIN {X 51.2431,Y -129.4498,Z 186,A -62.0867,B 2.9178,C 0.2971,E1 2.9966,E2 515.0554} C_DIS
LIN {X 54.8428,Y -127.965,Z 186,A -60.6181,B 2.9179,C 0.2963,E1 3.0004,E2 513.6041} C_DIS
LIN {X 57.6893,Y -126.709,Z 186,A -59.2259,B 2.9182,C 0.2937,E1 3.004,E2 512.1957} C_DIS
LIN {X 60.9493,Y -125.1729,Z 186,A -57.8056,B 2.9183,C 0.2922,E1 3.0075,E2 510.783} C_DIS
LIN {X 64.6431,Y -123.3038,Z 186,A -56.3038,B 2.9184,C 0.2915,E1 3.0112,E2 509.3075} C_DIS
LIN {X 68.3923,Y -121.2669,Z 186,A -54.5049,B 2.9187,C 0.2885,E1 3.0156,E2 507.5015} C_DIS
LIN {X 72.2794,Y -118.9911,Z 186,A -52.4321,B 2.9192,C 0.2836,E1 3.0206,E2 505.3973} C_DIS
LIN {X 75.3336,Y -117.0815,Z 186,A -51.278,B 2.9192,C 0.2841,E1 3.0233,E2 504.287} C_DIS
LIN {X 78.8472,Y -114.7442,Z 186,A -49.5555,B 2.9194,C 0.2813,E1 3.0272,E2 502.5651} C_DIS
LIN {X 82.2942,Y -112.2978,Z 186,A -47.9052,B 2.9196,C 0.279,E1 3.031,E2 500.9257} C_DIS
LIN {X 86.3209,Y -109.2336,Z 186,A -45.8646,B 2.92,C 0.2756,E1 3.0355,E2 498.8892} C_DIS
LIN {X 89.6977,Y -106.4777,Z 186,A -44.09,B 2.9203,C 0.2723,E1 3.0393,E2 497.1158} C_DIS
LIN {X 92.6983,Y -103.8759,Z 186,A -42.4849,B 2.9205,C 0.2694,E1 3.0426,E2 495.5134} C_DIS
LIN {X 96.3412,Y -100.5064,Z 186,A -40.5522,B 2.9208,C 0.2663,E1 3.0465,E2 493.5939} C_DIS
LIN {X 99.5446,Y -97.3346,Z 186,A -38.7684,B 2.9211,C 0.2631,E1 3.05,E2 491.8183} C_DIS
LIN {X 102.5301,Y -94.1843,Z 186,A -37.062,B 2.9214,C 0.26,E1 3.0533,E2 490.1213} C_DIS
LIN {X 105.7503,Y -90.5546,Z 186,A -35.0852,B 2.9218,C 0.2558,E1 3.0569,E2 488.1456} C_DIS
LIN {X 108.6632,Y -87.038,Z 186,A -33.2545,B 2.9221,C 0.252,E1 3.0601,E2 486.3199} C_DIS
LIN {X 110.8057,Y -84.2931,Z 186,A -31.5407,B 2.9226,C 0.246,E1 3.0631,E2 484.5669} C_DIS
LIN {X 113.4097,Y -80.7553,Z 186,A -30.1742,B 2.9226,C 0.246,E1 3.0652,E2 483.2588} C_DIS
LIN {X 115.3454,Y -77.9651,Z 186,A -28.7694,B 2.9229,C 0.2426,E1 3.0674,E2 481.8519} C_DIS
LIN {X 118.022,Y -73.8515,Z 186,A -26.8614,B 2.9232,C 0.2387,E1 3.0703,E2 479.9574} C_DIS
LIN {X 120.1829,Y -70.2798,Z 186,A -24.9867,B 2.9237,C 0.233,E1 3.073,E2 478.0601} C_DIS
LIN {X 122.0439,Y -66.9966,Z 186,A -23.7368,B 2.9237,C 0.232,E1 3.0746,E2 476.8498} C_DIS
LIN {X 123.8186,Y -63.6538,Z 186,A -22.331,B 2.9239,C 0.2295,E1 3.0764,E2 475.4631} C_DIS
LIN {X 125.4899,Y -60.2904,Z 186,A -20.8567,B 2.9242,C 0.2263,E1 3.0782,E2 473.9972} C_DIS
LIN {X 127.3816,Y -56.1872,Z 186,A -18.9657,B 2.9246,C 0.2211,E1 3.0804,E2 472.1006} C_DIS
LIN {X 128.9668,Y -52.4435,Z 186,A -17.4695,B 2.9248,C 0.2184,E1 3.0819,E2 470.6267} C_DIS
LIN {X 130.133,Y -49.4819,Z 186,A -16.3017,B 2.9249,C 0.2163,E1 3.0831,E2 469.4768} C_DIS
LIN {X 131.7206,Y -45.0841,Z 186,A -14.2996,B 2.9254,C 0.2104,E1 3.085,E2 467.4628} C_DIS
LIN {X 133.055,Y -40.9758,Z 186,A -12.6422,B 2.9256,C 0.2068,E1 3.0863,E2 465.8201} C_DIS
LIN {X 134.1735,Y -37.1511,Z 186,A -11.2767,B 2.9257,C 0.205,E1 3.0874,E2 464.4898} C_DIS
LIN {X 135.2715,Y -32.9293,Z 186,A -9.3666,B 2.9262,C 0.199,E1 3.0887,E2 462.5632} C_DIS
LIN {X 136.8254,Y -25.7222,Z 186,A -6.3998,B 2.9267,C 0.1912,E1 3.0904,E2 459.6032} C_DIS
LIN {X 137.3443,Y -22.7864,Z 186,A -5.1124,B 2.9269,C 0.1872,E1 3.091,E2 458.3071} C_DIS
LIN {X 137.9994,Y -18.4104,Z 186,A -3.5472,B 2.9271,C 0.1847,E1 3.0916,E2 456.7744} C_DIS
LIN {X 138.5151,Y -14.0277,Z 186,A -1.792,B 2.9274,C 0.1802,E1 3.0921,E2 455.0261} C_DIS
LIN {X 138.8435,Y -10.2569,Z 186,A -0.4004,B 2.9275,C 0.1774,E1 3.0924,E2 453.6552} C_DIS
LIN {X 139.0594,Y -6.7267,Z 186,A 1.0427,B 2.9278,C 0.1734,E1 3.0926,E2 452.2128} C_DIS
LIN {X 139.2009,Y -2.4148,Z 186,A 2.7178,B 2.928,C 0.1694,E1 3.0927,E2 450.5497} C_DIS
LIN {X 139.2049,Y 2.1737,Z 186,A 4.5025,B 2.9283,C 0.1651,E1 3.0927,E2 448.7773} C_DIS
LIN {X 139.0863,Y 6.188,Z 186,A 6.1709,B 2.9285,C 0.1603,E1 3.0925,E2 447.106} C_DIS
LIN {X 138.8541,Y 10.1108,Z 186,A 7.5986,B 2.9287,C 0.1576,E1 3.0923,E2 445.702} C_DIS
LIN {X 138.56,Y 13.5599,Z 186,A 8.9956,B 2.9289,C 0.1539,E1 3.0919,E2 444.3078} C_DIS
LIN {X 138.0791,Y 17.8021,Z 186,A 10.6454,B 2.9291,C 0.15,E1 3.0913,E2 442.6709} C_DIS
LIN {X 137.6014,Y 21.1784,Z 186,A 12.6092,B 2.9295,C 0.1406,E1 3.0905,E2 440.633} C_DIS
LIN {X 136.6746,Y 26.5113,Z 186,A 14.1672,B 2.9295,C 0.141,E1 3.0897,E2 439.1614} C_DIS
LIN {X 135.8188,Y 30.5952,Z 186,A 15.8164,B 2.9297,C 0.1369,E1 3.0887,E2 437.5201} C_DIS
LIN {X 134.9468,Y 34.2343,Z 186,A 17.178,B 2.9298,C 0.1344,E1 3.0878,E2 436.1808} C_DIS
LIN {X 133.9229,Y 38.0474,Z 186,A 18.8443,B 2.9301,C 0.1296,E1 3.0866,E2 434.5084} C_DIS
Enddeposition()
END
